KUKA KRL program: MyProgram_056().src

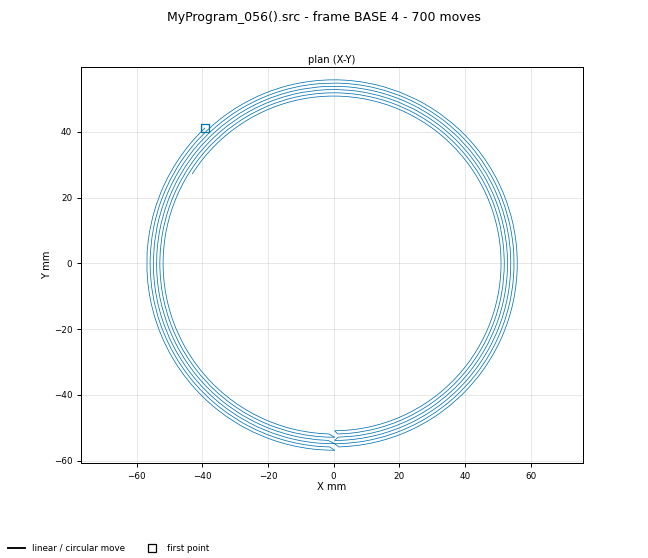
[picture p0: tool path of MyProgram_056().src in frame BASE 4, 700 of 700 moves have a stored position in this frame; points joined in program order, loops and branches not executed]
&ACCESS RVP
&REL 1
&PARAM TEMPLATE = C:\KRC\Roboter\Template\vorgabe
&PARAM EDITMASK = *
DEF MyProgram_056()
; ---- Setting reference (Base) ----
$BASE = BASE_DATA[4]

; --------------------------
; ---- Setting tool (TCP) ----
$TOOL = TOOL_DATA[3]
; --------------------------

$VEL.CP = VEL_APROX_PRINT
Startdeposition()
$VEL.CP = VEL_PRINT
LIN {X -39.2172,Y 41.1867,Z 69,A 127.6689,B 24.8602,C -2.7285,E1 24.8886,E2 316.0913} C_DIS
LIN {X -40.9874,Y 39.4246,Z 69,A 130.4028,B 24.8604,C -2.7263,E1 24.8832,E2 313.351} C_DIS
LIN {X -42.6349,Y 37.6376,Z 69,A 132.6601,B 24.8614,C -2.717,E1 24.879,E2 311.106} C_DIS
LIN {X -43.8253,Y 36.2439,Z 69,A 134.361,B 24.8621,C -2.7098,E1 24.876,E2 309.4144} C_DIS
LIN {X -45.2719,Y 34.4212,Z 69,A 137.1048,B 24.8621,C -2.7105,E1 24.8713,E2 306.656} C_DIS
LIN {X -46.7578,Y 32.3725,Z 69,A 139.4158,B 24.8631,C -2.6996,E1 24.8675,E2 304.3597} C_DIS
LIN {X -48.6669,Y 29.4246,Z 69,A 142.6739,B 24.8646,C -2.6851,E1 24.8627,E2 301.1198} C_DIS
LIN {X -50.461,Y 26.2306,Z 69,A 146.5624,B 24.8653,C -2.6778,E1 24.8574,E2 297.2282} C_DIS
LIN {X -51.6339,Y 23.8376,Z 69,A 149.8111,B 24.8652,C -2.6794,E1 24.8535,E2 293.9581} C_DIS
LIN {X -52.591,Y 21.6446,Z 69,A 152.047,B 24.8662,C -2.6693,E1 24.8511,E2 291.7339} C_DIS
LIN {X -54.117,Y 17.4819,Z 69,A 155.8039,B 24.8687,C -2.644,E1 24.8476,E2 288.0163} C_DIS
LIN {X -55.0295,Y 14.3546,Z 69,A 159.6144,B 24.8689,C -2.6425,E1 24.8446,E2 284.1872} C_DIS
LIN {X -55.9932,Y 9.9516,Z 69,A 164.0183,B 24.8705,C -2.6261,E1 24.8421,E2 279.7967} C_DIS
LIN {X -56.4492,Y 6.9116,Z 69,A 167.4164,B 24.871,C -2.6213,E1 24.8408,E2 276.3898} C_DIS
LIN {X -56.7032,Y 4.3633,Z 69,A 169.8052,B 24.8721,C -2.61,E1 24.8402,E2 274.0137} C_DIS
LIN {X -56.8029,Y 2.784,Z 69,A 172.173,B 24.8713,C -2.6178,E1 24.8398,E2 271.6129} C_DIS
LIN {X -56.832,Y -2.1175,Z 69,A 176.7138,B 24.8735,C -2.5956,E1 24.84,E2 267.0978} C_DIS
LIN {X -56.5731,Y -5.8044,Z 69,A -179.4639,B 24.8745,C -2.5856,E1 24.8409,E2 263.2765} C_DIS
LIN {X -56.1247,Y -9.1763,Z 69,A -175.6273,B 24.8748,C -2.5819,E1 24.8425,E2 259.4258} C_DIS
LIN {X -55.5073,Y -12.3803,Z 69,A -172.4836,B 24.8761,C -2.5695,E1 24.8443,E2 256.2933} C_DIS
LIN {X -54.4839,Y -16.303,Z 69,A -169.0489,B 24.8783,C -2.5464,E1 24.8468,E2 252.8938} C_DIS
LIN {X -53.1275,Y -20.2917,Z 69,A -164.2541,B 24.8786,C -2.5434,E1 24.8513,E2 248.0791} C_DIS
LIN {X -51.6778,Y -23.7434,Z 69,A -160.1585,B 24.879,C -2.5383,E1 24.8559,E2 243.973} C_DIS
LIN {X -49.9679,Y -27.1564,Z 69,A -155.8698,B 24.8793,C -2.5357,E1 24.8616,E2 239.6677} C_DIS
LIN {X -48.3498,Y -29.9434,Z 69,A -153.9425,B 24.8823,C -2.5045,E1 24.8643,E2 237.8052} C_DIS
LIN {X -47.405,Y -31.4172,Z 69,A -151.1609,B 24.881,C -2.5177,E1 24.8686,E2 234.978} C_DIS
LIN {X -45.5694,Y -34.0253,Z 69,A -148.4069,B 24.8825,C -2.5019,E1 24.8731,E2 232.2486} C_DIS
LIN {X -43.8437,Y -36.2217,Z 69,A -145.7476,B 24.8834,C -2.4926,E1 24.8777,E2 229.5989} C_DIS
LIN {X -42.1667,Y -38.1612,Z 69,A -143.2615,B 24.8841,C -2.4852,E1 24.8823,E2 227.1194} C_DIS
LIN {X -40.203,Y -40.2255,Z 69,A -140.3437,B 24.8846,C -2.48,E1 24.888,E2 224.2014} C_DIS
LIN {X -38.9195,Y -41.4673,Z 69,A -138.3237,B 24.8846,C -2.4803,E1 24.8921,E2 222.1723} C_DIS
LIN {X -36.6153,Y -43.5165,Z 69,A -135.3681,B 24.8853,C -2.4717,E1 24.8983,E2 219.2257} C_DIS
LIN {X -35.2522,Y -44.6267,Z 69,A -133.4026,B 24.8853,C -2.4721,E1 24.9026,E2 217.2521} C_DIS
LIN {X -32.9611,Y -46.3447,Z 69,A -130.6893,B 24.886,C -2.4641,E1 24.9087,E2 214.5482} C_DIS
LIN {X -30.637,Y -47.9129,Z 69,A -128.1623,B 24.887,C -2.4542,E1 24.9146,E2 212.0364} C_DIS
LIN {X -28.4476,Y -49.2444,Z 69,A -125.4187,B 24.887,C -2.4535,E1 24.9212,E2 209.286} C_DIS
LIN {X -27.09,Y -50.0039,Z 69,A -123.5686,B 24.8867,C -2.4567,E1 24.9257,E2 207.423} C_DIS
LIN {X -24.5055,Y -51.3202,Z 69,A -120.6332,B 24.887,C -2.4535,E1 24.9331,E2 204.4877} C_DIS
LIN {X -20.5017,Y -53.0469,Z 69,A -116.289,B 24.8875,C -2.4481,E1 24.9443,E2 200.1463} C_DIS
LIN {X -17.9953,Y -53.9487,Z 69,A -113.3864,B 24.8873,C -2.4502,E1 24.9519,E2 197.2333} C_DIS
LIN {X -14.7454,Y -54.9258,Z 69,A -110.05,B 24.8877,C -2.4464,E1 24.9609,E2 193.9007} C_DIS
LIN {X -11.3581,Y -55.7249,Z 69,A -106.2768,B 24.8873,C -2.45,E1 24.9712,E2 190.114} C_DIS
LIN {X -7.8896,Y -56.3208,Z 69,A -103.0939,B 24.8881,C -2.4419,E1 24.98,E2 186.9476} C_DIS
LIN {X -5.5019,Y -56.6045,Z 69,A -100.4271,B 24.8877,C -2.4465,E1 24.9874,E2 184.2682} C_DIS
LIN {X -1.8837,Y -56.8395,Z 69,A -97.1781,B 24.8884,C -2.4386,E1 24.9964,E2 181.0372} C_DIS
LIN {X 0.2942,Y -56.8688,Z 69,A -94.7619,B 24.8879,C -2.4436,E1 25.0032,E2 178.6091} C_DIS
Enddeposition()
LIN {X 0.2942,Y -56.8688,Z 69,A -94.7619,B 24.8879,C -2.4436,E1 25.0032,E2 178.6091} C_DIS
Startdeposition()
$VEL.CP = VEL_PRINT
LIN {X -1.1563,Y -55.8706,Z 69,A -97.7717,B 24.8892,C -2.4303,E1 24.9947,E2 181.6506} C_DIS
LIN {X -3.9674,Y -55.7418,Z 69,A -100.5256,B 24.8889,C -2.4327,E1 24.987,E2 184.3997} C_DIS
LIN {X -6.1298,Y -55.5461,Z 69,A -102.5576,B 24.8886,C -2.4366,E1 24.9814,E2 186.4236} C_DIS
LIN {X -8.8114,Y -55.184,Z 69,A -105.8724,B 24.8895,C -2.427,E1 24.9722,E2 189.7639} C_DIS
LIN {X -11.2153,Y -54.7455,Z 69,A -108.5068,B 24.8895,C -2.4256,E1 24.965,E2 192.4047} C_DIS
LIN {X -14.4657,Y -53.9778,Z 69,A -111.4901,B 24.8887,C -2.4357,E1 24.9569,E2 195.3683} C_DIS
LIN {X -17.2391,Y -53.1565,Z 69,A -114.2557,B 24.8881,C -2.4415,E1 24.9496,E2 198.1248} C_DIS
LIN {X -20.1585,Y -52.1197,Z 69,A -118.1024,B 24.889,C -2.4321,E1 24.9394,E2 202.0018} C_DIS
LIN {X -23.4557,Y -50.7217,Z 69,A -121.4951,B 24.8882,C -2.441,E1 24.9308,E2 205.3813} C_DIS
LIN {X -26.3548,Y -49.2786,Z 69,A -124.5245,B 24.8873,C -2.4504,E1 24.9233,E2 208.3968} C_DIS
LIN {X -28.2294,Y -48.2285,Z 69,A -127.0901,B 24.8876,C -2.447,E1 24.9171,E2 210.9781} C_DIS
LIN {X -32.493,Y -45.4648,Z 69,A -131.9283,B 24.8863,C -2.4616,E1 24.9059,E2 215.7973} C_DIS
LIN {X -34.8994,Y -43.6461,Z 69,A -134.9439,B 24.8856,C -2.4684,E1 24.8992,E2 218.8079} C_DIS
LIN {X -36.3752,Y -42.4229,Z 69,A -137.1316,B 24.8856,C -2.4682,E1 24.8945,E2 221.0044} C_DIS
LIN {X -38.2156,Y -40.7728,Z 69,A -139.6921,B 24.8852,C -2.4727,E1 24.8893,E2 223.5645} C_DIS
LIN {X -40.5593,Y -38.4426,Z 69,A -142.9215,B 24.8843,C -2.4825,E1 24.883,E2 226.7843} C_DIS
LIN {X -42.2441,Y -36.5828,Z 69,A -145.691,B 24.8841,C -2.4849,E1 24.8778,E2 229.5606} C_DIS
LIN {X -43.7711,Y -34.7412,Z 69,A -148.0469,B 24.8834,C -2.4922,E1 24.8737,E2 231.91} C_DIS
LIN {X -45.3492,Y -32.6552,Z 69,A -151.9009,B 24.8846,C -2.4794,E1 24.8673,E2 235.8134} C_DIS
LIN {X -47.2892,Y -29.7762,Z 69,A -154.1335,B 24.8817,C -2.5101,E1 24.864,E2 237.9838} C_DIS
LIN {X -49.316,Y -26.2841,Z 69,A -158.3271,B 24.8808,C -2.52,E1 24.8582,E2 242.1755} C_DIS
LIN {X -50.9281,Y -23.0038,Z 69,A -163.1438,B 24.8814,C -2.5131,E1 24.8524,E2 247.035} C_DIS
LIN {X -52.421,Y -19.3633,Z 69,A -166.7779,B 24.8797,C -2.531,E1 24.8488,E2 250.6466} C_DIS
LIN {X -53.4954,Y -16.1607,Z 69,A -170.252,B 24.8788,C -2.541,E1 24.8459,E2 254.1168} C_DIS
LIN {X -54.643,Y -11.7063,Z 69,A -175.3559,B 24.878,C -2.5491,E1 24.8426,E2 259.2312} C_DIS
LIN {X -55.4079,Y -7.2679,Z 69,A -179.6155,B 24.8761,C -2.569,E1 24.8408,E2 263.4687} C_DIS
LIN {X -55.8182,Y -2.6947,Z 69,A 176.0425,B 24.8741,C -2.5895,E1 24.8399,E2 267.7879} C_DIS
LIN {X -55.8798,Y 0.646,Z 69,A 171.9713,B 24.8741,C -2.5901,E1 24.8399,E2 271.882} C_DIS
LIN {X -55.7659,Y 3.6112,Z 69,A 168.9639,B 24.8731,C -2.6003,E1 24.8404,E2 274.8832} C_DIS
LIN {X -55.3001,Y 8.0451,Z 69,A 164.794,B 24.871,C -2.621,E1 24.8418,E2 279.0285} C_DIS
LIN {X -54.6598,Y 11.6265,Z 69,A 160.9401,B 24.8701,C -2.6307,E1 24.8438,E2 282.882} C_DIS
LIN {X -54.2027,Y 13.6015,Z 69,A 157.9464,B 24.8708,C -2.6229,E1 24.8459,E2 285.9119} C_DIS
LIN {X -53.2693,Y 16.892,Z 69,A 155.7786,B 24.8677,C -2.6546,E1 24.8476,E2 288.0163} C_DIS
LIN {X -52.4312,Y 19.3353,Z 69,A 152.3082,B 24.8682,C -2.6497,E1 24.8509,E2 291.5182} C_DIS
LIN {X -51.3497,Y 22.0459,Z 69,A 149.5456,B 24.8669,C -2.6622,E1 24.8538,E2 294.2662} C_DIS
LIN {X -49.6499,Y 25.6475,Z 69,A 145.2405,B 24.8661,C -2.6706,E1 24.8592,E2 298.5744} C_DIS
LIN {X -47.6251,Y 29.2363,Z 69,A 141.5872,B 24.8639,C -2.6916,E1 24.8642,E2 302.1963} C_DIS
LIN {X -46.6447,Y 30.7754,Z 69,A 139.4884,B 24.8638,C -2.6931,E1 24.8675,E2 304.3022} C_DIS
LIN {X -45.0843,Y 33.019,Z 69,A 136.7763,B 24.8629,C -2.7021,E1 24.8718,E2 307.0061} C_DIS
LIN {X -43.6194,Y 34.9328,Z 69,A 133.7277,B 24.8632,C -2.6991,E1 24.8772,E2 310.0762} C_DIS
LIN {X -41.8062,Y 37.0831,Z 69,A 130.8559,B 24.8624,C -2.7065,E1 24.8824,E2 312.9432} C_DIS
LIN {X -38.7269,Y 40.2875,Z 69,A 127.0324,B 24.8601,C -2.7294,E1 24.8899,E2 316.7284} C_DIS
LIN {X -36.5928,Y 42.2358,Z 69,A 123.7421,B 24.86,C -2.7306,E1 24.8967,E2 320.0289} C_DIS
LIN {X -34.5428,Y 43.9275,Z 69,A 121.0731,B 24.8593,C -2.7374,E1 24.9025,E2 322.6918} C_DIS
LIN {X -32.5769,Y 45.405,Z 69,A 118.0371,B 24.8596,C -2.7338,E1 24.9094,E2 325.747} C_DIS
LIN {X -29.9751,Y 47.1635,Z 69,A 114.8787,B 24.8589,C -2.7409,E1 24.9168,E2 328.8988} C_DIS
LIN {X -26.9091,Y 48.9779,Z 69,A 111.1784,B 24.8583,C -2.7463,E1 24.9258,E2 332.5968} C_DIS
LIN {X -23.4032,Y 50.7462,Z 69,A 107.9098,B 24.8563,C -2.7657,E1 24.9339,E2 335.8278} C_DIS
LIN {X -21.3454,Y 51.646,Z 69,A 104.8546,B 24.8574,C -2.7558,E1 24.9418,E2 338.9137} C_DIS
LIN {X -18.8923,Y 52.5928,Z 69,A 101.8682,B 24.8575,C -2.7541,E1 24.9497,E2 341.91} C_DIS
LIN {X -15.6131,Y 53.6579,Z 69,A 99.2156,B 24.8555,C -2.7736,E1 24.9566,E2 344.5207} C_DIS
LIN {X -13.6089,Y 54.201,Z 69,A 96.8585,B 24.8557,C -2.7716,E1 24.963,E2 346.8861} C_DIS
LIN {X -10.4708,Y 54.8928,Z 69,A 93.3705,B 24.8557,C -2.7709,E1 24.9726,E2 350.3799} C_DIS
LIN {X -7.2946,Y 55.4042,Z 69,A 90.2188,B 24.8553,C -2.7757,E1 24.9813,E2 353.5228} C_DIS
LIN {X -4.7136,Y 55.6839,Z 69,A 87.6823,B 24.8549,C -2.7793,E1 24.9883,E2 356.0521} C_DIS
LIN {X -1.6238,Y 55.8589,Z 69,A 84.0021,B 24.8558,C -2.771,E1 24.9986,E2 359.7529} C_DIS
LIN {X 1.2574,Y 55.8688,Z 69,A 81.6723,B 24.8545,C -2.7832,E1 25.005,E2 362.0536} C_DIS
LIN {X 3.3945,Y 55.7801,Z 69,A 79.203,B 24.855,C -2.778,E1 25.012,E2 364.5343} C_DIS
LIN {X 5.9454,Y 55.5654,Z 69,A 76.6605,B 24.855,C -2.7793,E1 25.019,E2 367.0722} C_DIS
LIN {X 8.4399,Y 55.2413,Z 69,A 73.5457,B 24.856,C -2.7684,E1 25.0277,E2 370.21} C_DIS
LIN {X 12.2895,Y 54.5152,Z 69,A 69.7213,B 24.8559,C -2.7703,E1 25.0381,E2 374.0252} C_DIS
LIN {X 15.2344,Y 53.7658,Z 69,A 66.4264,B 24.8564,C -2.7648,E1 25.047,E2 377.3277} C_DIS
LIN {X 20.1257,Y 52.1336,Z 69,A 60.752,B 24.8577,C -2.7525,E1 25.0619,E2 383.0196} C_DIS
LIN {X 25.3523,Y 49.8008,Z 69,A 56.0409,B 24.856,C -2.7689,E1 25.0737,E2 387.6796} C_DIS
LIN {X 27.2999,Y 48.7603,Z 69,A 53.3836,B 24.8571,C -2.7579,E1 25.0803,E2 390.3554} C_DIS
LIN {X 29.7779,Y 47.2881,Z 69,A 50.5649,B 24.8573,C -2.7563,E1 25.087,E2 393.169} C_DIS
LIN {X 32.2689,Y 45.6248,Z 69,A 47.4717,B 24.8579,C -2.7509,E1 25.0941,E2 396.2645} C_DIS
LIN {X 35.9602,Y 42.7763,Z 69,A 41.7497,B 24.8608,C -2.7228,E1 25.1066,E2 402.0317} C_DIS
LIN {X 38.4921,Y 40.5128,Z 69,A 39.3504,B 24.8592,C -2.7384,E1 25.1115,E2 404.3842} C_DIS
LIN {X 40.2273,Y 38.7893,Z 69,A 36.7009,B 24.86,C -2.7301,E1 25.1167,E2 407.0419} C_DIS
LIN {X 41.7484,Y 37.1477,Z 69,A 33.8256,B 24.8618,C -2.7127,E1 25.1221,E2 409.9455} C_DIS
LIN {X 44.1955,Y 34.1997,Z 69,A 30.3565,B 24.8618,C -2.7133,E1 25.1281,E2 413.3971} C_DIS
LIN {X 46.2331,Y 31.3904,Z 69,A 27.0938,B 24.862,C -2.7109,E1 25.1333,E2 416.6496} C_DIS
LIN {X 47.8397,Y 28.8832,Z 69,A 23.6663,B 24.8636,C -2.695,E1 25.1384,E2 420.0973} C_DIS
LIN {X 49.2731,Y 26.3647,Z 69,A 21.3439,B 24.863,C -2.7012,E1 25.1415,E2 422.393} C_DIS
LIN {X 50.2963,Y 24.3548,Z 69,A 18.6165,B 24.8645,C -2.6858,E1 25.1449,E2 425.1422} C_DIS
LIN {X 51.5199,Y 21.646,Z 69,A 15.6819,B 24.8652,C -2.6797,E1 25.1481,E2 428.0752} C_DIS
LIN {X 52.6763,Y 18.657,Z 69,A 12.175,B 24.8666,C -2.6654,E1 25.1515,E2 431.5963} C_DIS
LIN {X 53.9396,Y 14.6072,Z 69,A 8.4354,B 24.8666,C -2.666,E1 25.1545,E2 435.3132} C_DIS
LIN {X 54.5401,Y 12.1781,Z 69,A 5.4765,B 24.8682,C -2.6495,E1 25.1564,E2 438.294} C_DIS
LIN {X 55.146,Y 9.0438,Z 69,A 2.324,B 24.8689,C -2.6421,E1 25.158,E2 441.4454} C_DIS
LIN {X 55.5326,Y 6.2472,Z 69,A -0.3717,B 24.8694,C -2.6376,E1 25.1589,E2 444.136} C_DIS
LIN {X 55.7159,Y 4.3131,Z 69,A -2.5339,B 24.8704,C -2.6276,E1 25.1594,E2 446.309} C_DIS
LIN {X 55.863,Y 1.4879,Z 69,A -5.3121,B 24.871,C -2.6212,E1 25.1598,E2 449.0857} C_DIS
LIN {X 55.8667,Y -1.3509,Z 69,A -8.1564,B 24.8718,C -2.6135,E1 25.1597,E2 451.9314} C_DIS
LIN {X 55.7646,Y -3.6273,Z 69,A -10.6623,B 24.8729,C -2.6023,E1 25.1593,E2 454.4488} C_DIS
LIN {X 55.4267,Y -7.1224,Z 69,A -14.3164,B 24.8741,C -2.5897,E1 25.1582,E2 458.111} C_DIS
LIN {X 54.95,Y -10.168,Z 69,A -17.4113,B 24.8749,C -2.5813,E1 25.1567,E2 461.2078} C_DIS
LIN {X 54.3541,Y -12.9827,Z 69,A -20.3146,B 24.8757,C -2.5731,E1 25.1549,E2 464.1136} C_DIS
LIN {X 53.5755,Y -15.8904,Z 69,A -23.4014,B 24.8766,C -2.5635,E1 25.1526,E2 467.2053} C_DIS
LIN {X 52.7396,Y -18.4764,Z 69,A -26.1022,B 24.8773,C -2.5569,E1 25.1502,E2 469.9064} C_DIS
LIN {X 51.7541,Y -21.0798,Z 69,A -28.6565,B 24.8775,C -2.555,E1 25.1476,E2 472.4511} C_DIS
LIN {X 51.0194,Y -22.8012,Z 69,A -30.7415,B 24.8784,C -2.5456,E1 25.1452,E2 474.547} C_DIS
LIN {X 49.9671,Y -25.0237,Z 69,A -33.3288,B 24.8792,C -2.5367,E1 25.1421,E2 477.1414} C_DIS
LIN {X 48.5902,Y -27.6023,Z 69,A -36.3304,B 24.88,C -2.528,E1 25.138,E2 480.1479} C_DIS
LIN {X 46.3715,Y -31.1859,Z 69,A -40.6,B 24.8811,C -2.5171,E1 25.1316,E2 484.4217} C_DIS
LIN {X 44.0879,Y -34.3393,Z 69,A -45.025,B 24.883,C -2.4971,E1 25.1242,E2 488.8731} C_DIS
LIN {X 40.9939,Y -37.9792,Z 69,A -49.9441,B 24.8842,C -2.4843,E1 25.115,E2 493.8002} C_DIS
LIN {X 39.162,Y -39.8649,Z 69,A -52.61,B 24.8847,C -2.4786,E1 25.1097,E2 496.4685} C_DIS
LIN {X 35.4494,Y -43.2007,Z 69,A -56.8574,B 24.884,C -2.4857,E1 25.1009,E2 500.6822} C_DIS
LIN {X 32.2747,Y -45.6206,Z 69,A -61.0272,B 24.885,C -2.4756,E1 25.0916,E2 504.861} C_DIS
LIN {X 30.6447,Y -46.7308,Z 69,A -63.3151,B 24.8859,C -2.466,E1 25.0862,E2 507.1639} C_DIS
LIN {X 28.2516,Y -48.2156,Z 69,A -66.2026,B 24.8864,C -2.4607,E1 25.0793,E2 510.055} C_DIS
LIN {X 25.6538,Y -49.6467,Z 69,A -69.235,B 24.8868,C -2.4558,E1 25.0718,E2 513.0904} C_DIS
LIN {X 23.2862,Y -50.8005,Z 69,A -71.854,B 24.887,C -2.4533,E1 25.0652,E2 515.7086} C_DIS
LIN {X 21.2463,Y -51.6864,Z 69,A -73.9677,B 24.887,C -2.4534,E1 25.0598,E2 517.8169} C_DIS
LIN {X 19.0659,Y -52.5295,Z 69,A -76.5804,B 24.8877,C -2.4458,E1 25.0529,E2 520.4421} C_DIS
LIN {X 16.0148,Y -53.5387,Z 69,A -79.6071,B 24.8876,C -2.4474,E1 25.0449,E2 523.4594} C_DIS
LIN {X 13.6162,Y -54.1989,Z 69,A -82.4492,B 24.8884,C -2.4389,E1 25.0372,E2 526.3173} C_DIS
LIN {X 10.7969,Y -54.83,Z 69,A -85.4401,B 24.8887,C -2.4357,E1 25.029,E2 529.312} C_DIS
LIN {X 7.9269,Y -55.3174,Z 69,A -88.5389,B 24.8891,C -2.4314,E1 25.0204,E2 532.4181} C_DIS
LIN {X 4.0472,Y -55.7364,Z 69,A -92.2438,B 24.8887,C -2.4351,E1 25.0102,E2 536.1119} C_DIS
LIN {X 1.5438,Y -55.8611,Z 69,A -94.7599,B 24.8887,C -2.4353,E1 25.0031,E2 538.627} C_DIS
LIN {X 1.5438,Y -55.8611,Z 69,A -94.7599,B 24.8887,C -2.4353,E1 25.0031,E2 538.627} C_DIS
Enddeposition()
LIN {X 0.3078,Y -54.8889,Z 69,A -96.2149,B 24.8875,C -2.4488,E1 24.9992,E2 540.0498} C_DIS
Startdeposition()
$VEL.CP = VEL_PRINT
LIN {X 1.7607,Y -54.8662,Z 69,A -93.3221,B 24.885,C -2.4757,E1 25.0074,E2 537.0933} C_DIS
LIN {X 3.9415,Y -54.7525,Z 69,A -90.7379,B 24.8843,C -2.4828,E1 25.0147,E2 534.4935} C_DIS
LIN {X 7.7223,Y -54.3485,Z 69,A -87.2647,B 24.885,C -2.4753,E1 25.0242,E2 531.0407} C_DIS
LIN {X 9.8604,Y -54.0016,Z 69,A -84.9507,B 24.8847,C -2.4781,E1 25.0306,E2 528.7226} C_DIS
LIN {X 11.9507,Y -53.5783,Z 69,A -82.4136,B 24.884,C -2.4864,E1 25.0376,E2 526.1691} C_DIS
LIN {X 15.4117,Y -52.6869,Z 69,A -79.0152,B 24.8842,C -2.4835,E1 25.0467,E2 522.783} C_DIS
LIN {X 18.6024,Y -51.6463,Z 69,A -75.2256,B 24.8833,C -2.4937,E1 25.0568,E2 518.9766} C_DIS
LIN {X 21.3221,Y -50.5842,Z 69,A -72.2279,B 24.883,C -2.4969,E1 25.0645,E2 515.9781} C_DIS
LIN {X 24.1748,Y -49.2849,Z 69,A -69.2059,B 24.883,C -2.4968,E1 25.0721,E2 512.9643} C_DIS
LIN {X 26.237,Y -48.2184,Z 69,A -66.8758,B 24.8828,C -2.4989,E1 25.0779,E2 510.6357} C_DIS
LIN {X 28.0467,Y -47.1889,Z 69,A -64.5247,B 24.8821,C -2.5065,E1 25.0836,E2 508.2737} C_DIS
LIN {X 31.0827,Y -45.2476,Z 69,A -60.7065,B 24.8813,C -2.515,E1 25.0925,E2 504.4481} C_DIS
LIN {X 33.9481,Y -43.1385,Z 69,A -57.007,B 24.8806,C -2.5224,E1 25.1007,E2 500.7444} C_DIS
LIN {X 36.4763,Y -41.0232,Z 69,A -53.3254,B 24.8793,C -2.5353,E1 25.1085,E2 497.0468} C_DIS
LIN {X 38.4338,Y -39.1953,Z 69,A -50.8298,B 24.8793,C -2.5353,E1 25.1135,E2 494.5614} C_DIS
LIN {X 41.3629,Y -36.0902,Z 69,A -46.4665,B 24.8785,C -2.5443,E1 25.1218,E2 490.196} C_DIS
LIN {X 43.1893,Y -33.8837,Z 69,A -43.221,B 24.8772,C -2.5577,E1 25.1275,E2 486.934} C_DIS
LIN {X 44.5719,Y -32.0432,Z 69,A -41.0372,B 24.877,C -2.5593,E1 25.1311,E2 484.7569} C_DIS
LIN {X 46.1415,Y -29.7382,Z 69,A -38.2147,B 24.8764,C -2.5654,E1 25.1354,E2 481.9341} C_DIS
LIN {X 47.3793,Y -27.7245,Z 69,A -35.8771,B 24.8761,C -2.5695,E1 25.1388,E2 479.5988} C_DIS
LIN {X 48.4434,Y -25.8206,Z 69,A -33.5604,B 24.8753,C -2.5769,E1 25.1419,E2 477.2767} C_DIS
LIN {X 49.6171,Y -23.4861,Z 69,A -30.6085,B 24.8741,C -2.5899,E1 25.1455,E2 474.3099} C_DIS
LIN {X 50.7655,Y -20.8878,Z 69,A -27.5944,B 24.8731,C -2.5999,E1 25.1488,E2 471.2887} C_DIS
LIN {X 52.0732,Y -17.3725,Z 69,A -24.2272,B 24.8731,C -2.5996,E1 25.152,E2 467.9412} C_DIS
LIN {X 52.9785,Y -14.3761,Z 69,A -20.5472,B 24.8712,C -2.6189,E1 25.1548,E2 464.2366} C_DIS
LIN {X 53.6071,Y -11.8189,Z 69,A -18.1201,B 24.8711,C -2.6203,E1 25.1564,E2 461.8203} C_DIS
LIN {X 54.0364,Y -9.6677,Z 69,A -15.8429,B 24.8704,C -2.6272,E1 25.1576,E2 459.54} C_DIS
LIN {X 54.4752,Y -6.773,Z 69,A -12.2739,B 24.8683,C -2.6483,E1 25.1589,E2 455.942} C_DIS
LIN {X 54.7345,Y -4.1907,Z 69,A -9.8753,B 24.8681,C -2.6499,E1 25.1595,E2 453.554} C_DIS
LIN {X 54.8723,Y -1.5596,Z 69,A -6.9852,B 24.867,C -2.6617,E1 25.1598,E2 450.6531} C_DIS
LIN {X 54.8458,Y 2.304,Z 69,A -3.484,B 24.8669,C -2.6625,E1 25.1596,E2 447.1708} C_DIS
LIN {X 54.7404,Y 4.1161,Z 69,A -1.3599,B 24.8658,C -2.6736,E1 25.1592,E2 445.0333} C_DIS
LIN {X 54.4882,Y 6.6683,Z 69,A 1.2573,B 24.8651,C -2.6806,E1 25.1584,E2 442.415} C_DIS
LIN {X 54.1257,Y 9.1548,Z 69,A 3.939,B 24.8641,C -2.69,E1 25.1572,E2 439.7268} C_DIS
LIN {X 53.4716,Y 12.4172,Z 69,A 7.4354,B 24.863,C -2.701,E1 25.1551,E2 436.2246} C_DIS
LIN {X 52.1691,Y 17.0826,Z 69,A 12.0922,B 24.8624,C -2.7072,E1 25.1515,E2 431.5798} C_DIS
LIN {X 51.0317,Y 20.2273,Z 69,A 15.8576,B 24.8607,C -2.7233,E1 25.1479,E2 427.7974} C_DIS
LIN {X 50.1181,Y 22.3963,Z 69,A 18.4068,B 24.8598,C -2.7322,E1 25.145,E2 425.241} C_DIS
LIN {X 48.8935,Y 24.9562,Z 69,A 21.0676,B 24.8596,C -2.7337,E1 25.1417,E2 422.5909} C_DIS
LIN {X 47.8716,Y 26.8647,Z 69,A 23.5648,B 24.8585,C -2.7449,E1 25.1383,E2 420.0802} C_DIS
LIN {X 45.2681,Y 31.0531,Z 69,A 28.6967,B 24.8572,C -2.7576,E1 25.1306,E2 414.944} C_DIS
LIN {X 42.9422,Y 34.1965,Z 69,A 32.3528,B 24.8572,C -2.7582,E1 25.1245,E2 411.3039} C_DIS
LIN {X 41.2956,Y 36.1667,Z 69,A 35.1967,B 24.8561,C -2.7678,E1 25.1193,E2 408.4502} C_DIS
LIN {X 39.5234,Y 38.0958,Z 69,A 38.2528,B 24.8548,C -2.7805,E1 25.1134,E2 405.3773} C_DIS
LIN {X 38.0363,Y 39.5807,Z 69,A 40.5786,B 24.854,C -2.7878,E1 25.1087,E2 403.0439} C_DIS
LIN {X 35.3978,Y 41.9578,Z 69,A 43.8415,B 24.8542,C -2.7856,E1 25.1019,E2 399.7992} C_DIS
LIN {X 33.4341,Y 43.538,Z 69,A 46.2795,B 24.8542,C -2.7863,E1 25.0966,E2 397.3686} C_DIS
LIN {X 31.6124,Y 44.8793,Z 69,A 49.1464,B 24.8526,C -2.8007,E1 25.09,E2 394.4775} C_DIS
LIN {X 29.3934,Y 46.3629,Z 69,A 51.8524,B 24.8524,C -2.8034,E1 25.0837,E2 391.774} C_DIS
LIN {X 26.4972,Y 48.0768,Z 69,A 55.3096,B 24.852,C -2.8071,E1 25.0753,E2 388.3183} C_DIS
LIN {X 23.265,Y 49.7206,Z 69,A 59.3264,B 24.851,C -2.8164,E1 25.0652,E2 384.2902} C_DIS
LIN {X 19.9301,Y 51.1488,Z 69,A 62.7313,B 24.8514,C -2.8125,E1 25.0564,E2 380.9022} C_DIS
LIN {X 15.5305,Y 52.6517,Z 69,A 67.9223,B 24.8503,C -2.8231,E1 25.0426,E2 375.696} C_DIS
LIN {X 11.5436,Y 53.6671,Z 69,A 71.3235,B 24.8519,C -2.808,E1 25.0335,E2 372.3356} C_DIS
LIN {X 7.924,Y 54.3196,Z 69,A 75.915,B 24.8502,C -2.8238,E1 25.0208,E2 367.7113} C_DIS
LIN {X 4.5145,Y 54.7077,Z 69,A 79.6652,B 24.8498,C -2.8274,E1 25.0103,E2 363.9548} C_DIS
LIN {X 1.3244,Y 54.8792,Z 69,A 83.2942,B 24.8493,C -2.8327,E1 25.0002,E2 360.3141} C_DIS
LIN {X -3.88,Y 54.7573,Z 69,A 88.0508,B 24.8508,C -2.8182,E1 24.987,E2 355.5909} C_DIS
LIN {X -6.8588,Y 54.4645,Z 69,A 91.3565,B 24.8506,C -2.8198,E1 24.9778,E2 352.2793} C_DIS
LIN {X -10.3303,Y 53.9136,Z 69,A 94.7745,B 24.8514,C -2.8126,E1 24.9684,E2 348.8751} C_DIS
LIN {X -13.9339,Y 53.0962,Z 69,A 98.3306,B 24.8523,C -2.8037,E1 24.9588,E2 345.3355} C_DIS
LIN {X -16.8029,Y 52.2596,Z 69,A 102.1774,B 24.8513,C -2.8132,E1 24.9485,E2 341.4595} C_DIS
LIN {X -19.8881,Y 51.1653,Z 69,A 105.9499,B 24.8511,C -2.8151,E1 24.9386,E2 337.6746} C_DIS
LIN {X -23.327,Y 49.6911,Z 69,A 109.4649,B 24.8525,C -2.8025,E1 24.9297,E2 334.1811} C_DIS
LIN {X -26.7078,Y 47.9592,Z 69,A 112.9401,B 24.854,C -2.7875,E1 24.9212,E2 330.732} C_DIS
LIN {X -28.4749,Y 46.9315,Z 69,A 115.2888,B 24.854,C -2.7874,E1 24.9155,E2 328.3765} C_DIS
LIN {X -30.5546,Y 45.6056,Z 69,A 117.6775,B 24.8549,C -2.7794,E1 24.91,E2 325.9991} C_DIS
LIN {X -31.8468,Y 44.7121,Z 69,A 119.6825,B 24.8546,C -2.7823,E1 24.9054,E2 323.9801} C_DIS
LIN {X -34.3388,Y 42.8289,Z 69,A 122.709,B 24.8557,C -2.7716,E1 24.8987,E2 320.9682} C_DIS
LIN {X -35.8802,Y 41.5463,Z 69,A 125.3915,B 24.8552,C -2.7769,E1 24.893,E2 318.2626} C_DIS
LIN {X -37.9922,Y 39.6232,Z 69,A 128.3831,B 24.8559,C -2.7701,E1 24.8869,E2 315.2747} C_DIS
LIN {X -41.0217,Y 36.478,Z 69,A 132.2898,B 24.8581,C -2.7483,E1 24.8796,E2 311.4032} C_DIS
LIN {X -42.9179,Y 34.2272,Z 69,A 135.4369,B 24.8588,C -2.7417,E1 24.874,E2 308.2574} C_DIS
LIN {X -44.0004,Y 32.8231,Z 69,A 137.6357,B 24.8588,C -2.7425,E1 24.8702,E2 306.0461} C_DIS
LIN {X -45.9385,Y 30.0513,Z 69,A 140.9763,B 24.86,C -2.7298,E1 24.865,E2 302.7192} C_DIS
LIN {X -47.4868,Y 27.5398,Z 69,A 144.3758,B 24.8604,C -2.7263,E1 24.8601,E2 299.3104} C_DIS
LIN {X -48.6858,Y 25.3603,Z 69,A 146.8424,B 24.8614,C -2.7168,E1 24.8569,E2 296.8536} C_DIS
LIN {X -49.9946,Y 22.6704,Z 69,A 149.9843,B 24.8623,C -2.7079,E1 24.8532,E2 293.7157} C_DIS
LIN {X -50.9895,Y 20.3343,Z 69,A 153.5038,B 24.8617,C -2.714,E1 24.8495,E2 290.162} C_DIS
LIN {X -52.0973,Y 17.3009,Z 69,A 155.7269,B 24.8646,C -2.6853,E1 24.8476,E2 287.9948} C_DIS
LIN {X -53.1359,Y 13.7835,Z 69,A 159.661,B 24.8656,C -2.6752,E1 24.8446,E2 284.0621} C_DIS
LIN {X -53.7724,Y 11.0416,Z 69,A 163.1337,B 24.8656,C -2.6745,E1 24.8425,E2 280.5706} C_DIS
LIN {X -54.562,Y 6.0398,Z 69,A 168.8672,B 24.8666,C -2.6651,E1 24.8403,E2 274.8256} C_DIS
LIN {X -54.8906,Y 0.7075,Z 69,A 174.2152,B 24.8688,C -2.6438,E1 24.8398,E2 269.4962} C_DIS
LIN {X -54.856,Y -2.0706,Z 69,A 176.6815,B 24.8703,C -2.6278,E1 24.84,E2 267.0534} C_DIS
LIN {X -54.5965,Y -5.7103,Z 69,A -179.4363,B 24.8714,C -2.6171,E1 24.8409,E2 263.1734} C_DIS
LIN {X -54.1905,Y -8.7576,Z 69,A -176.0306,B 24.8721,C -2.6103,E1 24.8423,E2 259.7635} C_DIS
LIN {X -53.472,Y -12.415,Z 69,A -172.001,B 24.873,C -2.6008,E1 24.8447,E2 255.7331} C_DIS
LIN {X -52.5099,Y -16.0054,Z 69,A -168.5053,B 24.8747,C -2.583,E1 24.8473,E2 252.2596} C_DIS
LIN {X -51.6179,Y -18.6816,Z 69,A -165.4514,B 24.8754,C -2.5763,E1 24.8501,E2 249.2045} C_DIS
LIN {X -50.1777,Y -22.2634,Z 69,A -161.5159,B 24.8766,C -2.5633,E1 24.8544,E2 245.278} C_DIS
LIN {X -49.1146,Y -24.5187,Z 69,A -159.015,B 24.8775,C -2.5546,E1 24.8574,E2 242.7846} C_DIS
LIN {X -47.9585,Y -26.7092,Z 69,A -155.645,B 24.8769,C -2.5606,E1 24.862,E2 239.3823} C_DIS
LIN {X -46.2105,Y -29.6307,Z 69,A -151.9467,B 24.8775,C -2.554,E1 24.8675,E2 235.681} C_DIS
LIN {X -44.3108,Y -32.4028,Z 69,A -149.0708,B 24.8794,C -2.5349,E1 24.8721,E2 232.8368} C_DIS
LIN {X -42.4318,Y -34.8288,Z 69,A -145.471,B 24.8794,C -2.5341,E1 24.8784,E2 229.2219} C_DIS
LIN {X -40.0812,Y -37.5087,Z 69,A -142.1458,B 24.8809,C -2.5193,E1 24.8846,E2 225.9175} C_DIS
LIN {X -37.5117,Y -40.0784,Z 69,A -138.0935,B 24.8812,C -2.516,E1 24.8928,E2 221.8561} C_DIS
LIN {X -34.8443,Y -42.4189,Z 69,A -134.6015,B 24.8822,C -2.5054,E1 24.9002,E2 218.376} C_DIS
LIN {X -32.4215,Y -44.2971,Z 69,A -131.4233,B 24.8827,C -2.4995,E1 24.9072,E2 215.2003} C_DIS
LIN {X -29.1391,Y -46.5221,Z 69,A -127.2806,B 24.8833,C -2.4931,E1 24.9169,E2 211.0592} C_DIS
LIN {X -25.6169,Y -48.5507,Z 69,A -123.2779,B 24.8843,C -2.4831,E1 24.9266,E2 207.0687} C_DIS
LIN {X -22.7434,Y -49.9617,Z 69,A -119.608,B 24.8841,C -2.4852,E1 24.9359,E2 203.3844} C_DIS
LIN {X -18.579,Y -51.6553,Z 69,A -114.6712,B 24.8841,C -2.4852,E1 24.9487,E2 198.4368} C_DIS
LIN {X -14.8242,Y -52.855,Z 69,A -110.9239,B 24.885,C -2.4756,E1 24.9587,E2 194.7063} C_DIS
LIN {X -12.4145,Y -53.4722,Z 69,A -107.9508,B 24.8844,C -2.4813,E1 24.9668,E2 191.7154} C_DIS
LIN {X -9.7739,Y -54.0173,Z 69,A -105.7217,B 24.8856,C -2.4692,E1 24.9729,E2 189.5127} C_DIS
LIN {X -7.6072,Y -54.3648,Z 69,A -103.0373,B 24.8849,C -2.4761,E1 24.9803,E2 186.8095} C_DIS
LIN {X -5.0979,Y -54.6571,Z 69,A -100.7539,B 24.8856,C -2.4691,E1 24.9866,E2 184.5415} C_DIS
LIN {X -3.5839,Y -54.7774,Z 69,A -98.5019,B 24.8844,C -2.482,E1 24.993,E2 182.258} C_DIS
LIN {X 0.3078,Y -54.8889,Z 69,A -96.2142,B 24.8875,C -2.4485,E1 24.9992,E2 180.0498} C_DIS
Enddeposition()
LIN {X 0.3078,Y -54.8889,Z 69,A -96.2142,B 24.8875,C -2.4485,E1 24.9992,E2 180.0498} C_DIS
Startdeposition()
$VEL.CP = VEL_PRINT
LIN {X -1.7154,Y -53.879,Z 69,A -99.0876,B 24.8871,C -2.4521,E1 24.9912,E2 182.915} C_DIS
LIN {X -5.1888,Y -53.6564,Z 69,A -102.4391,B 24.8865,C -2.4586,E1 24.9819,E2 186.2527} C_DIS
LIN {X -9.2905,Y -53.1002,Z 69,A -106.0575,B 24.8851,C -2.4739,E1 24.972,E2 189.8378} C_DIS
LIN {X -11.4422,Y -52.6779,Z 69,A -109.0179,B 24.8861,C -2.4635,E1 24.9638,E2 192.8264} C_DIS
LIN {X -13.9646,Y -52.0661,Z 69,A -111.9395,B 24.8862,C -2.4622,E1 24.9559,E2 195.7554} C_DIS
LIN {X -17.614,Y -50.9476,Z 69,A -115.5787,B 24.8853,C -2.4726,E1 24.9463,E2 199.3764} C_DIS
LIN {X -20.1677,Y -49.9917,Z 69,A -118.5708,B 24.8852,C -2.4736,E1 24.9385,E2 202.3724} C_DIS
LIN {X -22.6816,Y -48.9023,Z 69,A -121.9621,B 24.8856,C -2.4686,E1 24.9298,E2 205.784} C_DIS
LIN {X -25.6061,Y -47.4365,Z 69,A -124.7535,B 24.8841,C -2.4846,E1 24.923,E2 208.5447} C_DIS
LIN {X -27.7915,Y -46.1906,Z 69,A -127.1949,B 24.8834,C -2.4923,E1 24.9171,E2 210.9752} C_DIS
LIN {X -29.188,Y -45.3205,Z 69,A -129.8388,B 24.8846,C -2.4798,E1 24.9108,E2 213.6572} C_DIS
LIN {X -32.5071,Y -43.0023,Z 69,A -133.7521,B 24.8833,C -2.4935,E1 24.902,E2 217.5517} C_DIS
LIN {X -34.1523,Y -41.7082,Z 69,A -136.4439,B 24.8836,C -2.4898,E1 24.8961,E2 220.2624} C_DIS
LIN {X -36.8078,Y -39.384,Z 69,A -139.8082,B 24.8824,C -2.5035,E1 24.8892,E2 223.6077} C_DIS
LIN {X -38.8716,Y -37.3482,Z 69,A -142.4922,B 24.8811,C -2.5163,E1 24.8839,E2 226.2723} C_DIS
LIN {X -40.8373,Y -35.1887,Z 69,A -145.9442,B 24.8811,C -2.5175,E1 24.8775,E2 229.737} C_DIS
LIN {X -42.36,Y -33.3396,Z 69,A -148.5735,B 24.8806,C -2.5221,E1 24.8729,E2 232.3676} C_DIS
LIN {X -43.9624,Y -31.1963,Z 69,A -151.7145,B 24.8804,C -2.5243,E1 24.8677,E2 235.5186} C_DIS
LIN {X -45.5595,Y -28.815,Z 69,A -154.155,B 24.8787,C -2.5415,E1 24.8641,E2 237.9303} C_DIS
LIN {X -47.4521,Y -25.5773,Z 69,A -158.365,B 24.8781,C -2.5485,E1 24.8582,E2 242.1456} C_DIS
LIN {X -48.7812,Y -22.9416,Z 69,A -161.7091,B 24.8776,C -2.5538,E1 24.8541,E2 245.495} C_DIS
LIN {X -50.0557,Y -20.0102,Z 69,A -164.9991,B 24.8765,C -2.5651,E1 24.8506,E2 248.7764} C_DIS
LIN {X -50.888,Y -17.7848,Z 69,A -167.8986,B 24.8763,C -2.5667,E1 24.8478,E2 251.6885} C_DIS
LIN {X -52.2722,Y -13.1742,Z 69,A -172.7439,B 24.8744,C -2.586,E1 24.8442,E2 256.5157} C_DIS
LIN {X -52.8826,Y -10.4588,Z 69,A -175.3048,B 24.873,C -2.601,E1 24.8427,E2 259.0558} C_DIS
LIN {X -53.2528,Y -8.3692,Z 69,A -177.8095,B 24.8727,C -2.6042,E1 24.8415,E2 261.5678} C_DIS
LIN {X -53.5694,Y -6.0201,Z 69,A 179.3301,B 24.8724,C -2.6068,E1 24.8405,E2 264.4391} C_DIS
LIN {X -53.8272,Y -2.9188,Z 69,A 176.1956,B 24.8711,C -2.6198,E1 24.8399,E2 267.5613} C_DIS
LIN {X -53.9039,Y -0.6033,Z 69,A 172.5162,B 24.8722,C -2.6094,E1 24.8399,E2 271.2877} C_DIS
LIN {X -53.8217,Y 3.0181,Z 69,A 170.3801,B 24.8684,C -2.6471,E1 24.8401,E2 273.3464} C_DIS
LIN {X -53.6164,Y 5.5825,Z 69,A 166.5664,B 24.8692,C -2.6395,E1 24.841,E2 277.2012} C_DIS
LIN {X -53.1026,Y 9.2771,Z 69,A 163.1502,B 24.8671,C -2.6602,E1 24.8425,E2 280.5884} C_DIS
LIN {X -52.4963,Y 12.2487,Z 69,A 159.6066,B 24.8666,C -2.6654,E1 24.8446,E2 284.1403} C_DIS
LIN {X -51.4612,Y 16.0509,Z 69,A 155.7238,B 24.8648,C -2.6829,E1 24.8476,E2 288.0037} C_DIS
LIN {X -50.2924,Y 19.4057,Z 69,A 152.0078,B 24.8636,C -2.6953,E1 24.8511,E2 291.7112} C_DIS
LIN {X -49.6061,Y 21.0986,Z 69,A 149.7734,B 24.8634,C -2.6966,E1 24.8535,E2 293.9549} C_DIS
LIN {X -48.1072,Y 24.3236,Z 69,A 146.2968,B 24.8618,C -2.7123,E1 24.8576,E2 297.4129} C_DIS
LIN {X -47.0768,Y 26.2612,Z 69,A 143.6451,B 24.8617,C -2.7141,E1 24.8612,E2 300.0743} C_DIS
LIN {X -45.2317,Y 29.3264,Z 69,A 139.4995,B 24.8611,C -2.7194,E1 24.8673,E2 304.2283} C_DIS
LIN {X -42.9118,Y 32.6263,Z 69,A 135.659,B 24.8592,C -2.7377,E1 24.8736,E2 308.0437} C_DIS
LIN {X -41.3716,Y 34.5585,Z 69,A 132.9787,B 24.8586,C -2.7436,E1 24.8783,E2 310.7223} C_DIS
LIN {X -39.8668,Y 36.2846,Z 69,A 130.375,B 24.8583,C -2.747,E1 24.8832,E2 313.3297} C_DIS
LIN {X -37.7891,Y 38.4432,Z 69,A 127.4504,B 24.8571,C -2.7586,E1 24.8889,E2 316.2388} C_DIS
LIN {X -36.2736,Y 39.8765,Z 69,A 124.9809,B 24.857,C -2.7597,E1 24.8939,E2 318.7159} C_DIS
LIN {X -34.1333,Y 41.7226,Z 69,A 121.7741,B 24.8566,C -2.763,E1 24.9008,E2 321.927} C_DIS
LIN {X -31.1167,Y 44.0192,Z 69,A 118.1632,B 24.8551,C -2.7779,E1 24.9089,E2 325.5152} C_DIS
LIN {X -28.7273,Y 45.6143,Z 69,A 114.5079,B 24.8555,C -2.7739,E1 24.9175,E2 329.192} C_DIS
LIN {X -26.5064,Y 46.9399,Z 69,A 112.2568,B 24.8541,C -2.7868,E1 24.9229,E2 331.4189} C_DIS
LIN {X -24.0029,Y 48.2675,Z 69,A 108.9731,B 24.8541,C -2.7872,E1 24.931,E2 334.7106} C_DIS
LIN {X -21.6166,Y 49.3821,Z 69,A 106.2218,B 24.8536,C -2.7921,E1 24.938,E2 337.457} C_DIS
LIN {X -19.0391,Y 50.4321,Z 69,A 103.6933,B 24.8524,C -2.8033,E1 24.9445,E2 339.9643} C_DIS
LIN {X -15.5514,Y 51.6148,Z 69,A 99.4884,B 24.8524,C -2.8029,E1 24.9557,E2 344.1778} C_DIS
LIN {X -12.8348,Y 52.356,Z 69,A 96.2302,B 24.8526,C -2.8013,E1 24.9645,E2 347.4447} C_DIS
LIN {X -9.7056,Y 53.0256,Z 69,A 92.3432,B 24.8532,C -2.7956,E1 24.9752,E2 351.3495} C_DIS
LIN {X -4.3993,Y 53.7265,Z 69,A 87.8841,B 24.8506,C -2.8204,E1 24.9875,E2 355.7524} C_DIS
LIN {X -2.409,Y 53.8525,Z 69,A 85.0985,B 24.8517,C -2.8093,E1 24.9953,E2 358.5653} C_DIS
LIN {X 1.3814,Y 53.8892,Z 69,A 81.5595,B 24.8507,C -2.8189,E1 25.0051,E2 362.0813} C_DIS
LIN {X 4.0072,Y 53.7579,Z 69,A 77.9297,B 24.8523,C -2.8037,E1 25.0153,E2 365.7458} C_DIS
LIN {X 6.4344,Y 53.5211,Z 69,A 75.505,B 24.8521,C -2.8063,E1 25.022,E2 368.1624} C_DIS
LIN {X 10.4156,Y 52.8909,Z 69,A 71.8374,B 24.851,C -2.8163,E1 25.032,E2 371.8025} C_DIS
LIN {X 12.8887,Y 52.3429,Z 69,A 68.5791,B 24.8523,C -2.8043,E1 25.041,E2 375.0848} C_DIS
LIN {X 15.7847,Y 51.5438,Z 69,A 65.4904,B 24.8523,C -2.804,E1 25.0492,E2 378.1688} C_DIS
LIN {X 18.6048,Y 50.5941,Z 69,A 62.5072,B 24.8523,C -2.8048,E1 25.0571,E2 381.1443} C_DIS
LIN {X 21.398,Y 49.4776,Z 69,A 59.1698,B 24.8529,C -2.7988,E1 25.0657,E2 384.4881} C_DIS
LIN {X 23.7463,Y 48.3942,Z 69,A 56.5494,B 24.8529,C -2.798,E1 25.0723,E2 387.1035} C_DIS
LIN {X 25.6912,Y 47.3904,Z 69,A 53.5903,B 24.8546,C -2.7827,E1 25.0796,E2 390.0907} C_DIS
LIN {X 28.6213,Y 45.6805,Z 69,A 50.5286,B 24.854,C -2.788,E1 25.0869,E2 393.13} C_DIS
LIN {X 31.0532,Y 44.0645,Z 69,A 47.4996,B 24.8544,C -2.7845,E1 25.0939,E2 396.1571} C_DIS
LIN {X 33.2159,Y 42.4577,Z 69,A 44.3845,B 24.8554,C -2.7744,E1 25.1008,E2 399.2846} C_DIS
LIN {X 36.7002,Y 39.4851,Z 69,A 39.7596,B 24.8559,C -2.77,E1 25.1105,E2 403.9018} C_DIS
LIN {X 38.1269,Y 38.1094,Z 69,A 37.126,B 24.8575,C -2.7549,E1 25.1157,E2 406.5601} C_DIS
LIN {X 41.2842,Y 34.6637,Z 69,A 32.7428,B 24.8574,C -2.7558,E1 25.1238,E2 410.9215} C_DIS
LIN {X 44.1966,Y 30.8635,Z 69,A 27.9595,B 24.858,C -2.7499,E1 25.1318,E2 415.6957} C_DIS
LIN {X 46.3741,Y 27.4833,Z 69,A 23.6787,B 24.8591,C -2.7389,E1 25.1382,E2 419.9811} C_DIS
LIN {X 48.1557,Y 24.2283,Z 69,A 19.8923,B 24.8599,C -2.7316,E1 25.1432,E2 423.7648} C_DIS
LIN {X 49.1007,Y 22.2489,Z 69,A 17.1886,B 24.8613,C -2.7173,E1 25.1464,E2 426.4878} C_DIS
LIN {X 50.4195,Y 19.0724,Z 69,A 13.373,B 24.8627,C -2.7035,E1 25.1504,E2 430.3149} C_DIS
LIN {X 51.5538,Y 15.7496,Z 69,A 9.1278,B 24.865,C -2.6817,E1 25.154,E2 434.5877} C_DIS
LIN {X 52.5476,Y 12.0267,Z 69,A 5.3783,B 24.8655,C -2.6767,E1 25.1565,E2 438.3273} C_DIS
LIN {X 53.2972,Y 8.0815,Z 69,A 1.3938,B 24.8662,C -2.6696,E1 25.1583,E2 442.3051} C_DIS
LIN {X 53.7216,Y 4.4607,Z 69,A -2.2728,B 24.8669,C -2.6621,E1 25.1594,E2 445.9679} C_DIS
LIN {X 53.9037,Y 0.6046,Z 69,A -6.888,B 24.8693,C -2.6382,E1 25.1598,E2 450.6122} C_DIS
LIN {X 53.8456,Y -2.5681,Z 69,A -9.4816,B 24.8687,C -2.6443,E1 25.1595,E2 453.1759} C_DIS
LIN {X 53.7071,Y -4.6377,Z 69,A -11.8084,B 24.8697,C -2.6347,E1 25.159,E2 455.5115} C_DIS
LIN {X 53.4417,Y -7.0628,Z 69,A -14.4737,B 24.8706,C -2.6249,E1 25.1581,E2 458.1841} C_DIS
LIN {X 53.1244,Y -9.1514,Z 69,A -16.4598,B 24.8708,C -2.6235,E1 25.1573,E2 460.162} C_DIS
LIN {X 52.7239,Y -11.2314,Z 69,A -18.9624,B 24.872,C -2.611,E1 25.1559,E2 462.6796} C_DIS
LIN {X 52.0968,Y -13.851,Z 69,A -21.8504,B 24.8729,C -2.6016,E1 25.1539,E2 465.5732} C_DIS
LIN {X 51.2708,Y -16.649,Z 69,A -24.5846,B 24.8731,C -2.5999,E1 25.1516,E2 468.2956} C_DIS
LIN {X 50.4601,Y -18.9638,Z 69,A -27.6767,B 24.8749,C -2.5816,E1 25.1487,E2 471.4139} C_DIS
LIN {X 49.5488,Y -21.2336,Z 69,A -30.3407,B 24.8758,C -2.5724,E1 25.1458,E2 474.085} C_DIS
LIN {X 47.9496,Y -24.6318,Z 69,A -33.6866,B 24.8756,C -2.5745,E1 25.1417,E2 477.4078} C_DIS
LIN {X 47.1618,Y -26.1089,Z 69,A -36.3651,B 24.8779,C -2.5503,E1 25.138,E2 480.1298} C_DIS
LIN {X 45.1402,Y -29.467,Z 69,A -39.8413,B 24.8776,C -2.5533,E1 25.1329,E2 483.5813} C_DIS
LIN {X 43.6193,Y -31.6746,Z 69,A -42.4302,B 24.8778,C -2.5511,E1 25.1288,E2 486.1626} C_DIS
LIN {X 41.6173,Y -34.2629,Z 69,A -46.0428,B 24.879,C -2.5391,E1 25.1225,E2 489.7866} C_DIS
LIN {X 40.2174,Y -35.895,Z 69,A -48.5004,B 24.8799,C -2.5298,E1 25.118,E2 492.2553} C_DIS
LIN {X 38.2721,Y -37.9624,Z 69,A -51.4554,B 24.8804,C -2.5237,E1 25.1123,E2 495.2118} C_DIS
LIN {X 36.7157,Y -39.4706,Z 69,A -53.8761,B 24.8812,C -2.5159,E1 25.1073,E2 497.6411} C_DIS
LIN {X 34.5482,Y -41.3801,Z 69,A -56.7051,B 24.8814,C -2.5141,E1 25.1013,E2 500.4634} C_DIS
LIN {X 32.3577,Y -43.1146,Z 69,A -59.7478,B 24.8821,C -2.5063,E1 25.0946,E2 503.5133} C_DIS
LIN {X 30.2527,Y -44.6168,Z 69,A -63.2407,B 24.884,C -2.4858,E1 25.0865,E2 507.043} C_DIS
LIN {X 27.6603,Y -46.2694,Z 69,A -66.3535,B 24.8843,C -2.4829,E1 25.0791,E2 510.1529} C_DIS
LIN {X 24.7098,Y -47.9098,Z 69,A -69.0899,B 24.8833,C -2.494,E1 25.0724,E2 512.8552} C_DIS
LIN {X 22.3391,Y -49.06,Z 69,A -72.4448,B 24.8847,C -2.4785,E1 25.0638,E2 516.2382} C_DIS
LIN {X 19.9813,Y -50.0671,Z 69,A -75.0926,B 24.8849,C -2.4762,E1 25.057,E2 518.8853} C_DIS
LIN {X 16.9848,Y -51.1611,Z 69,A -78.1611,B 24.8847,C -2.4783,E1 25.0489,E2 521.9426} C_DIS
LIN {X 14.2901,Y -51.9782,Z 69,A -81.2903,B 24.8853,C -2.4724,E1 25.0405,E2 525.0807} C_DIS
LIN {X 11.7465,Y -52.6115,Z 69,A -84.058,B 24.8855,C -2.4701,E1 25.033,E2 527.8499} C_DIS
LIN {X 8.9138,Y -53.1641,Z 69,A -87.0787,B 24.8856,C -2.4686,E1 25.0247,E2 530.8708} C_DIS
LIN {X 6.2311,Y -53.5449,Z 69,A -89.8538,B 24.8856,C -2.4688,E1 25.017,E2 533.6433} C_DIS
LIN {X 3.7289,Y -53.7772,Z 69,A -92.6237,B 24.8859,C -2.4656,E1 25.0093,E2 536.4192} C_DIS
LIN {X 1.5649,Y -53.8836,Z 69,A -94.5643,B 24.8853,C -2.4716,E1 25.0039,E2 538.345} C_DIS
LIN {X 0.3158,Y -53.8954,Z 69,A -96.302,B 24.8861,C -2.4638,E1 24.999,E2 540.1012} C_DIS
Enddeposition()
LIN {X 0.3158,Y -53.8954,Z 69,A -96.302,B 24.8861,C -2.4638,E1 24.999,E2 540.1012} C_DIS
Startdeposition()
$VEL.CP = VEL_PRINT
LIN {X 1.3078,Y -52.9029,Z 69,A -93.1346,B 24.8807,C -2.5205,E1 25.0082,E2 536.7996} C_DIS
LIN {X 6.1663,Y -52.5576,Z 69,A -88.9631,B 24.8825,C -2.5021,E1 25.0197,E2 532.6742} C_DIS
LIN {X 7.956,Y -52.3168,Z 69,A -86.2088,B 24.8809,C -2.5188,E1 25.0274,E2 529.8827} C_DIS
LIN {X 11.5199,Y -51.6496,Z 69,A -82.8773,B 24.8817,C -2.5105,E1 25.0365,E2 526.5748} C_DIS
LIN {X 13.9339,Y -51.0509,Z 69,A -79.7602,B 24.8806,C -2.5216,E1 25.045,E2 523.4363} C_DIS
LIN {X 16.2454,Y -50.3629,Z 69,A -77.4088,B 24.8808,C -2.5195,E1 25.0512,E2 521.0942} C_DIS
LIN {X 18.7314,Y -49.492,Z 69,A -74.5357,B 24.8805,C -2.5236,E1 25.0587,E2 518.2173} C_DIS
LIN {X 22.0056,Y -48.1261,Z 69,A -70.3898,B 24.8793,C -2.5353,E1 25.0694,E2 514.0536} C_DIS
LIN {X 24.7084,Y -46.7956,Z 69,A -67.3405,B 24.8793,C -2.5364,E1 25.077,E2 511.0102} C_DIS
LIN {X 27.0768,Y -45.4666,Z 69,A -64.6227,B 24.8792,C -2.5371,E1 25.0835,E2 508.299} C_DIS
LIN {X 29.6029,Y -43.8634,Z 69,A -61.552,B 24.8789,C -2.5398,E1 25.0907,E2 505.2319} C_DIS
LIN {X 31.3932,Y -42.6007,Z 69,A -58.9334,B 24.878,C -2.5497,E1 25.0967,E2 502.5991} C_DIS
LIN {X 34.0093,Y -40.5432,Z 69,A -55.0332,B 24.8766,C -2.5636,E1 25.1051,E2 498.6806} C_DIS
LIN {X 36.7819,Y -38.0451,Z 69,A -51.3216,B 24.8764,C -2.5661,E1 25.1127,E2 494.9784} C_DIS
LIN {X 38.6633,Y -36.1318,Z 69,A -48.441,B 24.8757,C -2.5726,E1 25.1183,E2 492.0948} C_DIS
LIN {X 41.0387,Y -33.409,Z 69,A -44.3754,B 24.8745,C -2.5858,E1 25.1257,E2 488.0164} C_DIS
LIN {X 42.6651,Y -31.3053,Z 69,A -41.7222,B 24.8742,C -2.5887,E1 25.1301,E2 485.3692} C_DIS
LIN {X 44.2113,Y -29.0808,Z 69,A -38.7362,B 24.8733,C -2.5978,E1 25.1348,E2 482.3763} C_DIS
LIN {X 45.6653,Y -26.7405,Z 69,A -35.6662,B 24.8723,C -2.6081,E1 25.1392,E2 479.2978} C_DIS
LIN {X 46.9393,Y -24.4355,Z 69,A -32.6285,B 24.8711,C -2.6203,E1 25.1432,E2 476.2471} C_DIS
LIN {X 48.7029,Y -20.6974,Z 69,A -29.0476,B 24.8717,C -2.6143,E1 25.1473,E2 472.6998} C_DIS
LIN {X 49.7724,Y -17.9739,Z 69,A -25.7313,B 24.8704,C -2.627,E1 25.1507,E2 469.3718} C_DIS
LIN {X 50.407,Y -16.1091,Z 69,A -23.2712,B 24.8691,C -2.6406,E1 25.1528,E2 466.8935} C_DIS
LIN {X 51.1637,Y -13.5164,Z 69,A -20.1522,B 24.8677,C -2.6539,E1 25.1552,E2 463.761} C_DIS
LIN {X 51.7305,Y -11.1488,Z 69,A -17.2816,B 24.8664,C -2.6673,E1 25.1569,E2 460.8755} C_DIS
LIN {X 52.2754,Y -8.2237,Z 69,A -14.5211,B 24.8664,C -2.6673,E1 25.1582,E2 458.131} C_DIS
LIN {X 52.6966,Y -4.8374,Z 69,A -10.4552,B 24.8644,C -2.6871,E1 25.1594,E2 454.0425} C_DIS
LIN {X 52.882,Y -1.9773,Z 69,A -7.2866,B 24.8633,C -2.6983,E1 25.1598,E2 450.8662} C_DIS
LIN {X 52.8538,Y 2.623,Z 69,A -2.7348,B 24.8626,C -2.7046,E1 25.1594,E2 446.3266} C_DIS
LIN {X 52.5509,Y 6.2238,Z 69,A 1.4162,B 24.8609,C -2.7219,E1 25.1583,E2 442.1591} C_DIS
LIN {X 51.8894,Y 10.3869,Z 69,A 5.9035,B 24.8596,C -2.7342,E1 25.1561,E2 437.6691} C_DIS
LIN {X 51.1355,Y 13.6207,Z 69,A 9.8728,B 24.8576,C -2.7531,E1 25.1533,E2 433.678} C_DIS
LIN {X 50.1235,Y 16.9696,Z 69,A 12.6024,B 24.8588,C -2.7415,E1 25.151,E2 430.9913} C_DIS
LIN {X 49.0271,Y 19.9166,Z 69,A 15.6467,B 24.8586,C -2.7436,E1 25.148,E2 427.9589} C_DIS
LIN {X 48.3588,Y 21.4901,Z 69,A 18.1465,B 24.8567,C -2.7626,E1 25.1452,E2 425.428} C_DIS
LIN {X 47.1393,Y 24.0461,Z 69,A 21.1583,B 24.8559,C -2.7698,E1 25.1415,E2 422.4152} C_DIS
LIN {X 45.8396,Y 26.4398,Z 69,A 23.6033,B 24.8562,C -2.767,E1 25.1382,E2 419.9895} C_DIS
LIN {X 44.9291,Y 27.9587,Z 69,A 26.4965,B 24.8535,C -2.7925,E1 25.1339,E2 417.0509} C_DIS
LIN {X 42.8752,Y 31.0177,Z 69,A 30.4435,B 24.8526,C -2.8014,E1 25.1276,E2 413.1021} C_DIS
LIN {X 41.1196,Y 33.3093,Z 69,A 33.1372,B 24.8528,C -2.7997,E1 25.1229,E2 410.4249} C_DIS
LIN {X 39.1077,Y 35.6503,Z 69,A 36.5899,B 24.8517,C -2.8094,E1 25.1165,E2 406.9647} C_DIS
LIN {X 37.5059,Y 37.3319,Z 69,A 38.9307,B 24.8516,C -2.8111,E1 25.1119,E2 404.6298} C_DIS
LIN {X 35.494,Y 39.2502,Z 69,A 42.2774,B 24.8502,C -2.824,E1 25.105,E2 401.2662} C_DIS
LIN {X 32.9966,Y 41.3716,Z 69,A 45.3085,B 24.8506,C -2.8201,E1 25.0986,E2 398.2559} C_DIS
LIN {X 31.0751,Y 42.8336,Z 69,A 48.1038,B 24.8497,C -2.8282,E1 25.0923,E2 395.4514} C_DIS
LIN {X 28.8406,Y 44.3694,Z 69,A 51.1047,B 24.8491,C -2.8341,E1 25.0853,E2 392.4465} C_DIS
LIN {X 25.4312,Y 46.4071,Z 69,A 54.8754,B 24.8496,C -2.8298,E1 25.0762,E2 388.6975} C_DIS
LIN {X 24.1847,Y 47.0685,Z 69,A 57.4104,B 24.8472,C -2.8514,E1 25.0698,E2 386.1181} C_DIS
LIN {X 19.5505,Y 49.1747,Z 69,A 61.831,B 24.8489,C -2.8362,E1 25.0586,E2 381.7444} C_DIS
LIN {X 16.8109,Y 50.177,Z 69,A 65.4607,B 24.8476,C -2.8479,E1 25.049,E2 378.0943} C_DIS
LIN {X 13.6668,Y 51.1231,Z 69,A 69.5864,B 24.8462,C -2.8611,E1 25.0379,E2 373.9439} C_DIS
LIN {X 9.674,Y 52.0273,Z 69,A 73.4777,B 24.8471,C -2.8529,E1 25.0273,E2 370.0772} C_DIS
LIN {X 6.7238,Y 52.4893,Z 69,A 76.3993,B 24.8476,C -2.848,E1 25.0193,E2 367.1698} C_DIS
LIN {X 5.0517,Y 52.6764,Z 69,A 79.2653,B 24.8455,C -2.8674,E1 25.0112,E2 364.2593} C_DIS
LIN {X 1.0678,Y 52.9074,Z 69,A 82.8579,B 24.847,C -2.8537,E1 25.0013,E2 360.7002} C_DIS
LIN {X -2.3403,Y 52.8664,Z 69,A 86.7809,B 24.8467,C -2.8569,E1 24.9903,E2 356.7692} C_DIS
LIN {X -4.9197,Y 52.689,Z 69,A 89.8193,B 24.8463,C -2.8598,E1 24.9818,E2 353.7222} C_DIS
LIN {X -9.6416,Y 52.0331,Z 69,A 94.1046,B 24.8484,C -2.8409,E1 24.9701,E2 349.4783} C_DIS
LIN {X -11.5101,Y 51.6517,Z 69,A 97.2476,B 24.8465,C -2.8579,E1 24.9614,E2 346.2908} C_DIS
LIN {X -15.1882,Y 50.6919,Z 69,A 100.5686,B 24.8485,C -2.8399,E1 24.9526,E2 343.0075} C_DIS
LIN {X -18.3529,Y 49.6342,Z 69,A 104.2682,B 24.8488,C -2.837,E1 24.9428,E2 339.3077} C_DIS
LIN {X -20.7487,Y 48.6813,Z 69,A 107.2708,B 24.8488,C -2.8367,E1 24.9351,E2 336.2991} C_DIS
LIN {X -23.6635,Y 47.3328,Z 69,A 110.854,B 24.8492,C -2.8331,E1 24.9261,E2 332.7152} C_DIS
LIN {X -26.0419,Y 46.0676,Z 69,A 113.5275,B 24.8502,C -2.8241,E1 24.9196,E2 330.0554} C_DIS
LIN {X -28.4994,Y 44.5884,Z 69,A 117.1053,B 24.8499,C -2.8262,E1 24.911,E2 326.4614} C_DIS
LIN {X -32.2018,Y 41.9927,Z 69,A 122.0018,B 24.851,C -2.8163,E1 24.9,E2 321.5712} C_DIS
LIN {X -35.0269,Y 39.6677,Z 69,A 125.7929,B 24.8522,C -2.8049,E1 24.892,E2 317.7927} C_DIS
LIN {X -37.5842,Y 37.2527,Z 69,A 129.086,B 24.854,C -2.7878,E1 24.8855,E2 314.5266} C_DIS
LIN {X -38.7028,Y 36.0896,Z 69,A 131.3598,B 24.8536,C -2.7919,E1 24.8811,E2 312.2331} C_DIS
LIN {X -41.1501,Y 33.2717,Z 69,A 135.0337,B 24.8553,C -2.7759,E1 24.8745,E2 308.5807} C_DIS
LIN {X -43.0363,Y 30.7931,Z 69,A 138.9485,B 24.8553,C -2.7754,E1 24.868,E2 304.6481} C_DIS
LIN {X -44.6134,Y 28.4605,Z 69,A 142.0237,B 24.8561,C -2.7674,E1 24.8633,E2 301.5764} C_DIS
LIN {X -46.7769,Y 24.7439,Z 69,A 146.3841,B 24.858,C -2.7496,E1 24.8574,E2 297.2358} C_DIS
LIN {X -47.995,Y 22.2892,Z 69,A 149.3847,B 24.8588,C -2.7415,E1 24.8538,E2 294.2384} C_DIS
LIN {X -49.1281,Y 19.6681,Z 69,A 152.4196,B 24.8599,C -2.7314,E1 24.8506,E2 291.2107} C_DIS
LIN {X -50.1349,Y 16.9359,Z 69,A 155.6237,B 24.8608,C -2.7226,E1 24.8476,E2 288.0094} C_DIS
LIN {X -50.9917,Y 14.1493,Z 69,A 159.3622,B 24.8608,C -2.7217,E1 24.8447,E2 284.2514} C_DIS
LIN {X -51.8542,Y 10.5584,Z 69,A 162.8371,B 24.863,C -2.7013,E1 24.8426,E2 280.8049} C_DIS
LIN {X -52.3249,Y 7.9038,Z 69,A 165.7788,B 24.8639,C -2.6925,E1 24.8413,E2 277.8668} C_DIS
LIN {X -52.7948,Y 3.6106,Z 69,A 170.1193,B 24.8659,C -2.6727,E1 24.8401,E2 273.5476} C_DIS
LIN {X -52.9175,Y 0.4058,Z 69,A 173.1717,B 24.8676,C -2.6554,E1 24.8398,E2 270.5181} C_DIS
LIN {X -52.9042,Y -1.2451,Z 69,A 175.7638,B 24.8669,C -2.6619,E1 24.8398,E2 267.895} C_DIS
LIN {X -52.7702,Y -3.9618,Z 69,A 178.7005,B 24.8679,C -2.6526,E1 24.8404,E2 264.963} C_DIS
LIN {X -52.4228,Y -7.2271,Z 69,A -177.4717,B 24.8686,C -2.6457,E1 24.8417,E2 261.1287} C_DIS
LIN {X -51.9881,Y -9.8785,Z 69,A -174.7356,B 24.8697,C -2.6342,E1 24.843,E2 258.4039} C_DIS
LIN {X -51.4219,Y -12.4946,Z 69,A -171.8297,B 24.8706,C -2.6255,E1 24.8448,E2 255.5016} C_DIS
LIN {X -50.5372,Y -15.6945,Z 69,A -168.211,B 24.8716,C -2.6153,E1 24.8477,E2 251.8866} C_DIS
LIN {X -49.6781,Y -18.2324,Z 69,A -165.3089,B 24.8724,C -2.6069,E1 24.8504,E2 248.9881} C_DIS
LIN {X -48.6698,Y -20.7759,Z 69,A -161.8474,B 24.8724,C -2.6063,E1 24.8541,E2 245.5088} C_DIS
LIN {X -47.0842,Y -24.154,Z 69,A -158.3919,B 24.8744,C -2.5861,E1 24.8583,E2 242.0828} C_DIS
LIN {X -45.9207,Y -26.2988,Z 69,A -155.6015,B 24.8749,C -2.5814,E1 24.8621,E2 239.2889} C_DIS
LIN {X -44.0413,Y -29.3382,Z 69,A -151.5355,B 24.8755,C -2.5747,E1 24.8682,E2 235.2183} C_DIS
LIN {X -42.3046,Y -31.7907,Z 69,A -148.2797,B 24.8763,C -2.5669,E1 24.8736,E2 231.9653} C_DIS
LIN {X -40.6543,Y -33.8757,Z 69,A -144.6349,B 24.8757,C -2.5728,E1 24.8801,E2 228.2898} C_DIS
LIN {X -37.6319,Y -37.2044,Z 69,A -140.6261,B 24.8781,C -2.5483,E1 24.8877,E2 224.322} C_DIS
LIN {X -35.648,Y -39.1099,Z 69,A -136.8412,B 24.8774,C -2.5558,E1 24.8956,E2 220.5039} C_DIS
LIN {X -32.4061,Y -41.8353,Z 69,A -133.0613,B 24.8795,C -2.534,E1 24.9037,E2 216.7617} C_DIS
LIN {X -30.2357,Y -43.4296,Z 69,A -129.2944,B 24.8785,C -2.5437,E1 24.9124,E2 212.9589} C_DIS
LIN {X -27.1864,Y -45.4017,Z 69,A -125.7194,B 24.8797,C -2.5318,E1 24.9209,E2 209.4011} C_DIS
LIN {X -23.8904,Y -47.2189,Z 69,A -121.8407,B 24.8805,C -2.5232,E1 24.9304,E2 205.5321} C_DIS
LIN {X -21.04,Y -48.5557,Z 69,A -118.6807,B 24.8813,C -2.5152,E1 24.9384,E2 202.3836} C_DIS
LIN {X -18.4767,Y -49.5885,Z 69,A -115.3659,B 24.881,C -2.5181,E1 24.9471,E2 199.0548} C_DIS
LIN {X -14.2355,Y -50.9678,Z 69,A -110.8402,B 24.8818,C -2.5092,E1 24.9592,E2 194.5423} C_DIS
LIN {X -11.6312,Y -51.6249,Z 69,A -107.5162,B 24.8812,C -2.5153,E1 24.9682,E2 191.1994} C_DIS
LIN {X -8.4833,Y -52.2337,Z 69,A -104.2608,B 24.8817,C -2.5103,E1 24.9772,E2 187.9528} C_DIS
LIN {X -4.9949,Y -52.682,Z 69,A -100.7961,B 24.8824,C -2.5034,E1 24.9867,E2 184.5021} C_DIS
LIN {X -1.9544,Y -52.8818,Z 69,A -97.3072,B 24.882,C -2.5071,E1 24.9965,E2 181.0035} C_DIS
LIN {X 0.3088,Y -52.91,Z 69,A -95.5075,B 24.8831,C -2.4956,E1 25.0015,E2 179.2311} C_DIS
Enddeposition()
LIN {X 0.3088,Y -52.91,Z 69,A -95.5075,B 24.8831,C -2.4956,E1 25.0015,E2 179.2311} C_DIS
Startdeposition()
$VEL.CP = VEL_PRINT
LIN {X -1.4817,Y -51.909,Z 69,A -98.3029,B 24.8829,C -2.4974,E1 24.9937,E2 182.0224} C_DIS
LIN {X -4.1613,Y -51.763,Z 69,A -101.1464,B 24.8827,C -2.4995,E1 24.9857,E2 184.862} C_DIS
LIN {X -7.0794,Y -51.4454,Z 69,A -104.7527,B 24.8833,C -2.4935,E1 24.9757,E2 188.485} C_DIS
LIN {X -10.2697,Y -50.9047,Z 69,A -108.0125,B 24.8827,C -2.5001,E1 24.9668,E2 191.7324} C_DIS
LIN {X -12.6548,Y -50.3653,Z 69,A -110.7271,B 24.8826,C -2.5012,E1 24.9594,E2 194.4482} C_DIS
LIN {X -14.508,Y -49.863,Z 69,A -112.8678,B 24.8825,C -2.5022,E1 24.9537,E2 196.5899} C_DIS
LIN {X -17.1117,Y -49.0298,Z 69,A -115.8948,B 24.8823,C -2.5044,E1 24.9456,E2 199.6173} C_DIS
LIN {X -19.4692,Y -48.1424,Z 69,A -118.6699,B 24.882,C -2.507,E1 24.9384,E2 202.3921} C_DIS
LIN {X -21.8328,Y -47.1176,Z 69,A -121.5226,B 24.8817,C -2.51,E1 24.9311,E2 205.2448} C_DIS
LIN {X -24.8834,Y -45.5803,Z 69,A -125.3302,B 24.8814,C -2.514,E1 24.9217,E2 209.0531} C_DIS
LIN {X -27.1189,Y -44.2868,Z 69,A -128.1396,B 24.8809,C -2.5187,E1 24.915,E2 211.8599} C_DIS
LIN {X -29.4161,Y -42.796,Z 69,A -131.1817,B 24.8805,C -2.5231,E1 24.9079,E2 214.9015} C_DIS
LIN {X -31.4905,Y -41.2934,Z 69,A -134.0822,B 24.8802,C -2.5267,E1 24.9014,E2 217.8037} C_DIS
LIN {X -34.1249,Y -39.1436,Z 69,A -138.0107,B 24.8798,C -2.5309,E1 24.893,E2 221.7374} C_DIS
LIN {X -36.495,Y -36.9437,Z 69,A -141.4372,B 24.8789,C -2.5403,E1 24.8861,E2 225.1557} C_DIS
LIN {X -38.0127,Y -35.3813,Z 69,A -144.6694,B 24.8796,C -2.5328,E1 24.8799,E2 228.42} C_DIS
LIN {X -40.4838,Y -32.5245,Z 69,A -148.1245,B 24.8776,C -2.5531,E1 24.8738,E2 231.8425} C_DIS
LIN {X -42.2055,Y -30.2562,Z 69,A -151.1552,B 24.8767,C -2.5623,E1 24.8688,E2 234.8658} C_DIS
LIN {X -43.9202,Y -27.7092,Z 69,A -154.5163,B 24.8759,C -2.5712,E1 24.8636,E2 238.2225} C_DIS
LIN {X -45.215,Y -25.542,Z 69,A -157.3848,B 24.8753,C -2.5772,E1 24.8596,E2 241.0915} C_DIS
LIN {X -46.3719,Y -23.3764,Z 69,A -160.8375,B 24.8757,C -2.5736,E1 24.8552,E2 244.5714} C_DIS
LIN {X -48.0948,Y -19.5862,Z 69,A -164.6527,B 24.8733,C -2.5979,E1 24.851,E2 248.3497} C_DIS
LIN {X -48.9999,Y -17.1969,Z 69,A -167.4008,B 24.8724,C -2.607,E1 24.8484,E2 251.0914} C_DIS
LIN {X -49.5509,Y -15.5391,Z 69,A -169.5594,B 24.8722,C -2.6093,E1 24.8465,E2 253.2569} C_DIS
LIN {X -50.2721,Y -13.0175,Z 69,A -172.3994,B 24.8712,C -2.6187,E1 24.8444,E2 256.091} C_DIS
LIN {X -50.8445,Y -10.5632,Z 69,A -175.2025,B 24.8704,C -2.6268,E1 24.8428,E2 258.8912} C_DIS
LIN {X -51.2959,Y -8.0922,Z 69,A -177.788,B 24.8693,C -2.638,E1 24.8415,E2 261.4653} C_DIS
LIN {X -51.6032,Y -5.8215,Z 69,A 179.4715,B 24.8689,C -2.6427,E1 24.8406,E2 264.2108} C_DIS
LIN {X -51.8231,Y -3.3349,Z 69,A 176.69,B 24.868,C -2.6509,E1 24.84,E2 266.9894} C_DIS
LIN {X -51.9247,Y -0.7662,Z 69,A 174.1022,B 24.8668,C -2.6634,E1 24.8398,E2 269.563} C_DIS
LIN {X -51.9104,Y 1.4363,Z 69,A 171.303,B 24.8666,C -2.6658,E1 24.8399,E2 272.3734} C_DIS
LIN {X -51.7906,Y 3.8151,Z 69,A 168.4781,B 24.866,C -2.6712,E1 24.8404,E2 275.2023} C_DIS
LIN {X -51.468,Y 6.9165,Z 69,A 165.3014,B 24.8645,C -2.6858,E1 24.8415,E2 278.3631} C_DIS
LIN {X -51.0529,Y 9.5093,Z 69,A 162.3015,B 24.8638,C -2.6934,E1 24.8429,E2 281.3626} C_DIS
LIN {X -50.4708,Y 12.2244,Z 69,A 159.4932,B 24.8624,C -2.7066,E1 24.8446,E2 284.1558} C_DIS
LIN {X -49.9131,Y 14.3333,Z 69,A 156.873,B 24.862,C -2.711,E1 24.8466,E2 286.7808} C_DIS
LIN {X -49.1536,Y 16.7534,Z 69,A 154.3061,B 24.8608,C -2.7229,E1 24.8487,E2 289.334} C_DIS
LIN {X -48.1116,Y 19.5449,Z 69,A 150.6745,B 24.8603,C -2.7278,E1 24.8524,E2 292.9741} C_DIS
LIN {X -47.0597,Y 21.957,Z 69,A 147.7779,B 24.8594,C -2.7364,E1 24.8557,E2 295.8659} C_DIS
LIN {X -45.88,Y 24.3265,Z 69,A 145.2775,B 24.8579,C -2.751,E1 24.8589,E2 298.3449} C_DIS
LIN {X -44.617,Y 26.5722,Z 69,A 142.0379,B 24.8576,C -2.7532,E1 24.8634,E2 301.5961} C_DIS
LIN {X -43.4045,Y 28.5093,Z 69,A 139.3362,B 24.8572,C -2.7575,E1 24.8675,E2 304.3011} C_DIS
LIN {X -41.2833,Y 31.5036,Z 69,A 135.5345,B 24.8557,C -2.7719,E1 24.8737,E2 308.0869} C_DIS
LIN {X -39.3606,Y 33.8734,Z 69,A 132.0442,B 24.855,C -2.7787,E1 24.8799,E2 311.5771} C_DIS
LIN {X -37.3773,Y 36.0508,Z 69,A 128.072,B 24.8553,C -2.7758,E1 24.8875,E2 315.5736} C_DIS
LIN {X -33.7194,Y 39.4935,Z 69,A 123.5922,B 24.8523,C -2.8044,E1 24.8967,E2 320.0031} C_DIS
LIN {X -32.0661,Y 40.8475,Z 69,A 120.6767,B 24.8526,C -2.8009,E1 24.903,E2 322.938} C_DIS
LIN {X -29.4037,Y 42.8046,Z 69,A 117.1214,B 24.8517,C -2.8095,E1 24.9111,E2 326.485} C_DIS
LIN {X -27.2641,Y 44.1982,Z 69,A 114.2618,B 24.8512,C -2.8141,E1 24.9178,E2 329.3429} C_DIS
LIN {X -24.9249,Y 45.5578,Z 69,A 111.2089,B 24.8508,C -2.8181,E1 24.9253,E2 332.395} C_DIS
LIN {X -22.0215,Y 47.0297,Z 69,A 107.6986,B 24.8501,C -2.825,E1 24.934,E2 335.898} C_DIS
LIN {X -19.6525,Y 48.0678,Z 69,A 104.8282,B 24.8497,C -2.8288,E1 24.9414,E2 338.7661} C_DIS
LIN {X -17.9771,Y 48.7195,Z 69,A 102.9196,B 24.8493,C -2.8325,E1 24.9464,E2 340.6697} C_DIS
LIN {X -14.2113,Y 49.9477,Z 69,A 98.4132,B 24.849,C -2.8352,E1 24.9584,E2 345.1776} C_DIS
LIN {X -11.6733,Y 50.601,Z 69,A 95.5406,B 24.8487,C -2.8382,E1 24.9662,E2 348.047} C_DIS
LIN {X -9.0405,Y 51.1373,Z 69,A 91.8583,B 24.8497,C -2.8286,E1 24.9764,E2 351.7561} C_DIS
LIN {X -5.0684,Y 51.6829,Z 69,A 88.377,B 24.8477,C -2.8469,E1 24.9859,E2 355.1961} C_DIS
LIN {X -2.1761,Y 51.8844,Z 69,A 85.0028,B 24.8479,C -2.8452,E1 24.9953,E2 358.5756} C_DIS
LIN {X 0.2948,Y 51.9292,Z 69,A 82.2049,B 24.8479,C -2.8445,E1 25.0031,E2 361.375} C_DIS
LIN {X 2.4907,Y 51.8709,Z 69,A 79.7037,B 24.8481,C -2.8433,E1 25.0101,E2 363.8783} C_DIS
LIN {X 5.8204,Y 51.6033,Z 69,A 76.147,B 24.8479,C -2.8452,E1 25.02,E2 367.4285} C_DIS
LIN {X 8.3323,Y 51.2577,Z 69,A 73.3039,B 24.8481,C -2.8437,E1 25.0278,E2 370.2727} C_DIS
LIN {X 10.9032,Y 50.7728,Z 69,A 70.7787,B 24.8475,C -2.849,E1 25.0347,E2 372.7822} C_DIS
LIN {X 12.7271,Y 50.3467,Z 69,A 68.3159,B 24.8484,C -2.8406,E1 25.0414,E2 375.2613} C_DIS
LIN {X 15.1634,Y 49.6674,Z 69,A 65.6068,B 24.8484,C -2.8402,E1 25.0487,E2 377.9669} C_DIS
LIN {X 17.55,Y 48.8753,Z 69,A 62.7098,B 24.8489,C -2.8356,E1 25.0564,E2 380.8689} C_DIS
LIN {X 19.3605,Y 48.1866,Z 69,A 59.4297,B 24.8514,C -2.8125,E1 25.065,E2 384.1963} C_DIS
LIN {X 22.696,Y 46.7084,Z 69,A 56.6254,B 24.8495,C -2.8304,E1 25.0719,E2 386.951} C_DIS
LIN {X 24.9523,Y 45.5429,Z 69,A 53.5989,B 24.8503,C -2.8225,E1 25.0794,E2 389.9876} C_DIS
LIN {X 27.5712,Y 44.0064,Z 69,A 50.5273,B 24.8503,C -2.8229,E1 25.0867,E2 393.0486} C_DIS
LIN {X 29.6925,Y 42.6038,Z 69,A 47.7205,B 24.8508,C -2.8183,E1 25.0932,E2 395.8567} C_DIS
LIN {X 31.7697,Y 41.0782,Z 69,A 44.9032,B 24.8513,C -2.8139,E1 25.0995,E2 398.6743} C_DIS
LIN {X 33.9204,Y 39.3221,Z 69,A 41.7543,B 24.852,C -2.8065,E1 25.1062,E2 401.8286} C_DIS
LIN {X 35.9648,Y 37.4602,Z 69,A 38.7474,B 24.8526,C -2.8013,E1 25.1123,E2 404.8356} C_DIS
LIN {X 37.8091,Y 35.5978,Z 69,A 36.1887,B 24.8526,C -2.8017,E1 25.1173,E2 407.3823} C_DIS
LIN {X 39.3009,Y 33.9448,Z 69,A 33.4876,B 24.8536,C -2.7914,E1 25.1223,E2 410.0958} C_DIS
LIN {X 40.8554,Y 32.0562,Z 69,A 30.8826,B 24.8541,C -2.787,E1 25.1269,E2 412.699} C_DIS
LIN {X 42.297,Y 30.128,Z 69,A 28.2181,B 24.8548,C -2.7804,E1 25.1313,E2 415.3663} C_DIS
LIN {X 43.5712,Y 28.2539,Z 69,A 25.4932,B 24.8559,C -2.7696,E1 25.1355,E2 418.1032} C_DIS
LIN {X 45.0791,Y 25.7802,Z 69,A 22.1325,B 24.8571,C -2.7579,E1 25.1402,E2 421.4742} C_DIS
LIN {X 46.6377,Y 22.8411,Z 69,A 18.8104,B 24.8574,C -2.755,E1 25.1444,E2 424.7856} C_DIS
LIN {X 47.7277,Y 20.4669,Z 69,A 15.8758,B 24.8584,C -2.7459,E1 25.1478,E2 427.7258} C_DIS
LIN {X 48.7064,Y 18.0129,Z 69,A 12.5014,B 24.8602,C -2.7282,E1 25.1511,E2 431.1233} C_DIS
LIN {X 49.8751,Y 14.467,Z 69,A 8.9061,B 24.8604,C -2.7268,E1 25.1541,E2 434.7015} C_DIS
LIN {X 50.6561,Y 11.4349,Z 69,A 5.1836,B 24.862,C -2.7108,E1 25.1565,E2 438.4401} C_DIS
LIN {X 51.4569,Y 7.0008,Z 69,A 0.5469,B 24.8628,C -2.7025,E1 25.1586,E2 443.0694} C_DIS
LIN {X 51.7528,Y 4.2897,Z 69,A -2.4128,B 24.8637,C -2.6942,E1 25.1594,E2 446.0312} C_DIS
LIN {X 51.9277,Y 0.5913,Z 69,A -6.928,B 24.8659,C -2.6724,E1 25.1598,E2 450.571} C_DIS
LIN {X 51.883,Y -2.2086,Z 69,A -10.1146,B 24.8671,C -2.6606,E1 25.1594,E2 453.7664} C_DIS
LIN {X 51.4663,Y -6.9286,Z 69,A -14.6095,B 24.8671,C -2.6594,E1 25.1581,E2 458.2377} C_DIS
LIN {X 50.8315,Y -10.6264,Z 69,A -18.8057,B 24.8686,C -2.6452,E1 25.156,E2 462.4429} C_DIS
LIN {X 50.2198,Y -13.2202,Z 69,A -21.7877,B 24.8696,C -2.6352,E1 25.154,E2 465.4314} C_DIS
LIN {X 49.4854,Y -15.7474,Z 69,A -24.5458,B 24.8702,C -2.6293,E1 25.1517,E2 468.1877} C_DIS
LIN {X 48.6396,Y -18.1924,Z 69,A -27.6033,B 24.8715,C -2.6164,E1 25.1488,E2 471.2585} C_DIS
LIN {X 47.4078,Y -21.1955,Z 69,A -31.1427,B 24.8724,C -2.6066,E1 25.1449,E2 474.8017} C_DIS
LIN {X 45.9262,Y -24.2387,Z 69,A -34.569,B 24.8729,C -2.6021,E1 25.1407,E2 478.2204} C_DIS
LIN {X 44.7091,Y -26.4163,Z 69,A -37.4128,B 24.8738,C -2.5924,E1 25.1367,E2 481.0724} C_DIS
LIN {X 43.3403,Y -28.6068,Z 69,A -40.2558,B 24.8746,C -2.5846,E1 25.1324,E2 483.9196} C_DIS
LIN {X 41.8469,Y -30.7501,Z 69,A -43.178,B 24.8754,C -2.576,E1 25.1276,E2 486.8478} C_DIS
LIN {X 40.4596,Y -32.5543,Z 69,A -45.71,B 24.8761,C -2.5691,E1 25.1233,E2 489.3845} C_DIS
LIN {X 38.6709,Y -34.6596,Z 69,A -48.6991,B 24.8767,C -2.5626,E1 25.1178,E2 492.3756} C_DIS
LIN {X 36.7565,Y -36.6846,Z 69,A -51.7571,B 24.8774,C -2.5555,E1 25.1118,E2 495.4372} C_DIS
LIN {X 34.7705,Y -38.5716,Z 69,A -54.4536,B 24.8774,C -2.555,E1 25.1063,E2 498.1237} C_DIS
LIN {X 33.4701,Y -39.7058,Z 69,A -56.6702,B 24.8785,C -2.5445,E1 25.1016,E2 500.3565} C_DIS
LIN {X 31.2889,Y -41.4457,Z 69,A -59.6874,B 24.879,C -2.5393,E1 25.0949,E2 503.3751} C_DIS
LIN {X 29.1944,Y -42.9467,Z 69,A -62.4819,B 24.8794,C -2.5346,E1 25.0885,E2 506.1711} C_DIS
LIN {X 26.3897,Y -44.7248,Z 69,A -66.6174,B 24.8809,C -2.5186,E1 25.0786,E2 510.3314} C_DIS
LIN {X 23.5732,Y -46.2713,Z 69,A -69.9315,B 24.8811,C -2.5172,E1 25.0704,E2 513.6396} C_DIS
LIN {X 20.7174,Y -47.6184,Z 69,A -73.1653,B 24.8811,C -2.5167,E1 25.0622,E2 516.8664} C_DIS
LIN {X 18.2521,Y -48.617,Z 69,A -76.1302,B 24.8815,C -2.5121,E1 25.0545,E2 519.8356} C_DIS
LIN {X 15.7688,Y -49.4785,Z 69,A -78.5891,B 24.8811,C -2.517,E1 25.048,E2 522.2782} C_DIS
LIN {X 13.7039,Y -50.0895,Z 69,A -81.3629,B 24.882,C -2.5069,E1 25.0406,E2 525.0713} C_DIS
LIN {X 11.276,Y -50.6915,Z 69,A -84.2533,B 24.8825,C -2.5019,E1 25.0327,E2 527.9696} C_DIS
LIN {X 7.5633,Y -51.377,Z 69,A -87.8781,B 24.8819,C -2.5087,E1 25.0228,E2 531.5743} C_DIS
LIN {X 4.9002,Y -51.6985,Z 69,A -91.8154,B 24.8837,C -2.4892,E1 25.0117,E2 535.5553} C_DIS
LIN {X 1.1935,Y -51.9169,Z 69,A -96.0571,B 24.8841,C -2.4852,E1 24.9998,E2 539.8055} C_DIS
LIN {X 1.1935,Y -51.9169,Z 69,A -96.0571,B 24.8841,C -2.4852,E1 24.9998,E2 539.8055} C_DIS
Enddeposition()
LIN {X 0.3002,Y -50.939,Z 69,A -95.324,B 24.8796,C -2.533,E1 25.0022,E2 538.9589} C_DIS
Startdeposition()
$VEL.CP = VEL_PRINT
LIN {X 2.4904,Y -50.8819,Z 69,A -92.5166,B 24.8789,C -2.54,E1 25.0101,E2 536.1356} C_DIS
LIN {X 4.9651,Y -50.7002,Z 69,A -89.7133,B 24.8787,C -2.5416,E1 25.0179,E2 533.3299} C_DIS
LIN {X 7.3885,Y -50.4038,Z 69,A -86.9608,B 24.8786,C -2.5435,E1 25.0255,E2 530.5752} C_DIS
LIN {X 9.911,Y -49.9693,Z 69,A -84.1146,B 24.8784,C -2.5452,E1 25.0333,E2 527.7282} C_DIS
LIN {X 12.3172,Y -49.431,Z 69,A -81.3524,B 24.8782,C -2.5476,E1 25.0408,E2 524.9641} C_DIS
LIN {X 14.6508,Y -48.79,Z 69,A -78.5779,B 24.8778,C -2.5516,E1 25.0483,E2 522.1849} C_DIS
LIN {X 17.1565,Y -47.9669,Z 69,A -75.6699,B 24.8775,C -2.5541,E1 25.056,E2 519.2767} C_DIS
LIN {X 19.4831,Y -47.0699,Z 69,A -72.8741,B 24.8772,C -2.5579,E1 25.0632,E2 516.4783} C_DIS
LIN {X 21.7618,Y -46.0607,Z 69,A -70.0923,B 24.8768,C -2.5617,E1 25.0703,E2 513.6944} C_DIS
LIN {X 23.9938,Y -44.9384,Z 69,A -67.292,B 24.8764,C -2.5662,E1 25.0772,E2 510.8914} C_DIS
LIN {X 26.2906,Y -43.6339,Z 69,A -64.3227,B 24.8759,C -2.5714,E1 25.0844,E2 507.9185} C_DIS
LIN {X 28.5915,Y -42.1617,Z 69,A -61.2627,B 24.8753,C -2.5771,E1 25.0916,E2 504.8553} C_DIS
LIN {X 30.5646,Y -40.7539,Z 69,A -58.6127,B 24.8749,C -2.5812,E1 25.0975,E2 502.205} C_DIS
LIN {X 32.5521,Y -39.1847,Z 69,A -55.7058,B 24.8742,C -2.5885,E1 25.1039,E2 499.2918} C_DIS
LIN {X 34.5459,Y -37.439,Z 69,A -52.7343,B 24.8736,C -2.5951,E1 25.11,E2 496.3165} C_DIS
LIN {X 36.3631,Y -35.6768,Z 69,A -49.8686,B 24.8729,C -2.6022,E1 25.1157,E2 493.446} C_DIS
LIN {X 38.2493,Y -33.6468,Z 69,A -46.7941,B 24.8722,C -2.6091,E1 25.1215,E2 490.3688} C_DIS
LIN {X 39.9327,Y -31.6301,Z 69,A -43.828,B 24.8714,C -2.617,E1 25.1267,E2 487.3979} C_DIS
LIN {X 41.448,Y -29.6166,Z 69,A -41.0633,B 24.8708,C -2.6232,E1 25.1313,E2 484.6319} C_DIS
LIN {X 42.8488,Y -27.551,Z 69,A -38.2341,B 24.87,C -2.6313,E1 25.1356,E2 481.7975} C_DIS
LIN {X 44.1467,Y -25.4195,Z 69,A -35.4338,B 24.8692,C -2.6391,E1 25.1396,E2 478.9931} C_DIS
LIN {X 45.3651,Y -23.1752,Z 69,A -32.6963,B 24.8687,C -2.6446,E1 25.1432,E2 476.2571} C_DIS
LIN {X 46.3966,Y -21.0344,Z 69,A -30.0656,B 24.868,C -2.6516,E1 25.1463,E2 473.6239} C_DIS
LIN {X 47.4312,Y -18.5839,Z 69,A -27.0037,B 24.8669,C -2.6621,E1 25.1495,E2 470.5543} C_DIS
LIN {X 48.2609,Y -16.3085,Z 69,A -24.2984,B 24.8661,C -2.67,E1 25.152,E2 467.8454} C_DIS
LIN {X 49.0208,Y -13.8577,Z 69,A -21.4322,B 24.8653,C -2.6785,E1 25.1543,E2 464.9756} C_DIS
LIN {X 49.6402,Y -11.4424,Z 69,A -18.687,B 24.8645,C -2.686,E1 25.1561,E2 462.2285} C_DIS
LIN {X 50.1333,Y -9.0403,Z 69,A -15.914,B 24.8636,C -2.6949,E1 25.1576,E2 459.4506} C_DIS
LIN {X 50.5132,Y -6.595,Z 69,A -13.1115,B 24.8627,C -2.7041,E1 25.1587,E2 456.6429} C_DIS
LIN {X 50.7791,Y -4.069,Z 69,A -10.3198,B 24.8619,C -2.7117,E1 25.1594,E2 453.8496} C_DIS
LIN {X 50.9189,Y -1.531,Z 69,A -7.5284,B 24.8611,C -2.7193,E1 25.1598,E2 451.0568} C_DIS
LIN {X 50.9394,Y 0.6021,Z 69,A -5.0625,B 24.8602,C -2.7283,E1 25.1598,E2 448.5845} C_DIS
LIN {X 50.8469,Y 3.1261,Z 69,A -2.3039,B 24.8595,C -2.7355,E1 25.1594,E2 445.8253} C_DIS
LIN {X 50.6335,Y 5.6056,Z 69,A 0.513,B 24.8585,C -2.7445,E1 25.1586,E2 443.0036} C_DIS
LIN {X 50.2995,Y 8.0701,Z 69,A 3.2905,B 24.8577,C -2.7528,E1 25.1574,E2 440.223} C_DIS
LIN {X 49.8465,Y 10.5107,Z 69,A 6.0789,B 24.8568,C -2.7612,E1 25.1559,E2 437.4309} C_DIS
LIN {X 49.2614,Y 12.9802,Z 69,A 8.8993,B 24.856,C -2.7691,E1 25.154,E2 434.6082} C_DIS
LIN {X 48.5684,Y 15.3714,Z 69,A 11.6806,B 24.8552,C -2.7769,E1 25.1517,E2 431.8241} C_DIS
LIN {X 47.7602,Y 17.7236,Z 69,A 14.4719,B 24.8543,C -2.7849,E1 25.1491,E2 429.0295} C_DIS
LIN {X 46.8223,Y 20.0712,Z 69,A 17.2861,B 24.8535,C -2.7924,E1 25.1461,E2 426.2133} C_DIS
LIN {X 45.7837,Y 22.3389,Z 69,A 20.0741,B 24.8528,C -2.7997,E1 25.1428,E2 423.4229} C_DIS
LIN {X 44.6247,Y 24.5724,Z 69,A 22.8801,B 24.852,C -2.8068,E1 25.1391,E2 420.6148} C_DIS
LIN {X 43.4113,Y 26.6569,Z 69,A 25.6037,B 24.8512,C -2.8141,E1 25.1352,E2 417.8879} C_DIS
LIN {X 42.0252,Y 28.7931,Z 69,A 28.4287,B 24.8506,C -2.8205,E1 25.1308,E2 415.0619} C_DIS
LIN {X 40.5828,Y 30.7924,Z 69,A 31.212,B 24.8498,C -2.8274,E1 25.1262,E2 412.2755} C_DIS
LIN {X 38.9813,Y 32.7968,Z 69,A 34.061,B 24.8492,C -2.8333,E1 25.1211,E2 409.4257} C_DIS
LIN {X 37.3186,Y 34.677,Z 69,A 36.8683,B 24.8486,C -2.8392,E1 25.1158,E2 406.6169} C_DIS
LIN {X 35.4774,Y 36.5577,Z 69,A 39.8395,B 24.8479,C -2.8456,E1 25.11,E2 403.6432} C_DIS
LIN {X 33.5142,Y 38.3651,Z 69,A 42.8041,B 24.8473,C -2.8507,E1 25.1038,E2 400.6783} C_DIS
LIN {X 31.5849,Y 39.9684,Z 69,A 45.6334,B 24.8468,C -2.856,E1 25.0976,E2 397.8471} C_DIS
LIN {X 29.7031,Y 41.3863,Z 69,A 48.3175,B 24.8462,C -2.8612,E1 25.0916,E2 395.1603} C_DIS
LIN {X 27.5535,Y 42.8472,Z 69,A 51.2066,B 24.8458,C -2.8651,E1 25.0849,E2 392.2715} C_DIS
LIN {X 25.4226,Y 44.1449,Z 69,A 54.0132,B 24.8453,C -2.8691,E1 25.0781,E2 389.4639} C_DIS
LIN {X 23.155,Y 45.3754,Z 69,A 56.8161,B 24.8451,C -2.871,E1 25.0712,E2 386.6644} C_DIS
LIN {X 20.9157,Y 46.4501,Z 69,A 59.6409,B 24.8447,C -2.8748,E1 25.064,E2 383.8378} C_DIS
LIN {X 18.5909,Y 47.4284,Z 69,A 62.4754,B 24.8444,C -2.8776,E1 25.0567,E2 381.0031} C_DIS
LIN {X 16.3147,Y 48.2588,Z 69,A 65.1952,B 24.8442,C -2.8798,E1 25.0495,E2 378.2835} C_DIS
LIN {X 13.8637,Y 49.0192,Z 69,A 68.0771,B 24.844,C -2.8818,E1 25.0418,E2 375.4019} C_DIS
LIN {X 11.4274,Y 49.6437,Z 69,A 70.8633,B 24.8439,C -2.8826,E1 25.0343,E2 372.6179} C_DIS
LIN {X 9.0562,Y 50.1305,Z 69,A 73.6223,B 24.8437,C -2.8843,E1 25.0267,E2 369.8579} C_DIS
LIN {X 6.5938,Y 50.5134,Z 69,A 76.4632,B 24.8435,C -2.8857,E1 25.0188,E2 367.0163} C_DIS
LIN {X 4.0457,Y 50.781,Z 69,A 79.3042,B 24.8435,C -2.8853,E1 25.011,E2 364.1779} C_DIS
LIN {X 1.5272,Y 50.919,Z 69,A 82.104,B 24.8437,C -2.8844,E1 25.0032,E2 361.381} C_DIS
LIN {X -0.8933,Y 50.9341,Z 69,A 84.9062,B 24.8436,C -2.8852,E1 24.9953,E2 358.5768} C_DIS
LIN {X -3.4542,Y 50.8247,Z 69,A 87.757,B 24.8438,C -2.8836,E1 24.9874,E2 355.7291} C_DIS
LIN {X -5.8821,Y 50.6012,Z 69,A 90.537,B 24.8438,C -2.8828,E1 24.9797,E2 352.9493} C_DIS
LIN {X -8.3705,Y 50.2495,Z 69,A 93.3677,B 24.844,C -2.881,E1 24.9719,E2 350.1205} C_DIS
LIN {X -10.721,Y 49.8012,Z 69,A 96.0852,B 24.8442,C -2.8792,E1 24.9644,E2 347.4041} C_DIS
LIN {X -13.3049,Y 49.1738,Z 69,A 99.0225,B 24.8447,C -2.8755,E1 24.9565,E2 344.4714} C_DIS
LIN {X -15.6207,Y 48.4879,Z 69,A 101.7853,B 24.8449,C -2.8732,E1 24.9491,E2 341.7093} C_DIS
LIN {X -17.9642,Y 47.6694,Z 69,A 104.5752,B 24.8453,C -2.8696,E1 24.9418,E2 338.9223} C_DIS
LIN {X -20.3847,Y 46.6856,Z 69,A 107.4969,B 24.8458,C -2.8652,E1 24.9343,E2 336.0043} C_DIS
LIN {X -22.6026,Y 45.6531,Z 69,A 110.2953,B 24.8461,C -2.8618,E1 24.9273,E2 333.207} C_DIS
LIN {X -24.8692,Y 44.459,Z 69,A 113.1393,B 24.8467,C -2.8564,E1 24.9203,E2 330.3679} C_DIS
LIN {X -27.0124,Y 43.1904,Z 69,A 115.9228,B 24.8473,C -2.851,E1 24.9137,E2 327.5884} C_DIS
LIN {X -29.0309,Y 41.8604,Z 69,A 118.733,B 24.8477,C -2.8472,E1 24.9072,E2 324.7779} C_DIS
LIN {X -31.0691,Y 40.3707,Z 69,A 121.615,B 24.8483,C -2.8421,E1 24.9007,E2 321.8979} C_DIS
LIN {X -33.1685,Y 38.6647,Z 69,A 124.6025,B 24.849,C -2.8346,E1 24.8944,E2 318.9167} C_DIS
LIN {X -35.1048,Y 36.9163,Z 69,A 127.552,B 24.8497,C -2.8282,E1 24.8883,E2 315.9707} C_DIS
LIN {X -36.9602,Y 35.0581,Z 69,A 130.5907,B 24.8504,C -2.8224,E1 24.8824,E2 312.9327} C_DIS
LIN {X -38.7041,Y 33.1223,Z 69,A 133.5079,B 24.8511,C -2.8149,E1 24.877,E2 310.0203} C_DIS
LIN {X -40.1595,Y 31.3431,Z 69,A 136.0729,B 24.8519,C -2.8079,E1 24.8726,E2 307.46} C_DIS
LIN {X -41.6364,Y 29.3525,Z 69,A 138.8769,B 24.8526,C -2.8007,E1 24.868,E2 304.6594} C_DIS
LIN {X -43.0103,Y 27.2994,Z 69,A 141.6696,B 24.8534,C -2.7933,E1 24.8638,E2 301.8705} C_DIS
Enddeposition()
END
